LIN {X 0,Y 510.056,Z 394.446,A -85,B 0,C 180,E1 -5580.789,E2 -5580.789} C_VEL
LIN {X 0,Y 509.95,Z 394.463,A -85,B 0,C 180,E1 -5583.16,E2 -5583.16} C_VEL
LIN {X 0,Y 509.969,Z 394.456,A -85,B 0,C 180,E1 -5586.329,E2 -5586.329} C_VEL
LIN {X 0,Y 509.909,Z 394.465,A -85,B 0,C 180,E1 -5588.72,E2 -5588.72} C_VEL
LIN {X 0,Y 509.894,Z 394.466,A -85,B 0,C 180,E1 -5591.931,E2 -5591.931} C_VEL
LIN {X 0,Y 509.883,Z 394.475,A -85,B 0,C 180,E1 -5595.242,E2 -5595.242} C_VEL
LIN {X 0,Y 509.879,Z 394.467,A -85,B 0,C 180,E1 -5598.001,E2 -5598.001} C_VEL
LIN {X 0,Y 509.841,Z 394.479,A -85,B 0,C 180,E1 -5601.002,E2 -5601.002} C_VEL
LIN {X 0,Y 509.86,Z 394.471,A -85,B 0,C 180,E1 -5604.426,E2 -5604.426} C_VEL
LIN {X 0,Y 509.878,Z 394.476,A -85,B 0,C 180,E1 -5607.055,E2 -5607.055} C_VEL
LIN {X 0,Y 509.871,Z 394.469,A -85,B 0,C 180,E1 -5609.75,E2 -5609.75} C_VEL
LIN {X 0,Y 509.868,Z 394.475,A -85,B 0,C 180,E1 -5612.775,E2 -5612.775} C_VEL
LIN {X 0,Y 509.834,Z 394.474,A -85,B 0,C 180,E1 -5615.581,E2 -5615.581} C_VEL
LIN {X 0,Y 509.85,Z 394.473,A -85,B 0,C 180,E1 -5618.337,E2 -5618.337} C_VEL
LIN {X 0,Y 509.857,Z 394.471,A -85,B 0,C 180,E1 -5621.425,E2 -5621.425} C_VEL
LIN {X 0,Y 509.848,Z 394.479,A -85,B 0,C 180,E1 -5624.668,E2 -5624.668} C_VEL
LIN {X 0,Y 509.853,Z 394.472,A -85,B 0,C 180,E1 -5628.103,E2 -5628.103} C_VEL
LIN {X 0,Y 509.84,Z 394.481,A -85,B 0,C 180,E1 -5630.648,E2 -5630.648} C_VEL
LIN {X 0,Y 509.825,Z 394.474,A -85,B 0,C 180,E1 -5633.744,E2 -5633.744} C_VEL
LIN {X 0,Y 509.159,Z 394.564,A -85,B 0,C 180,E1 -5634.404,E2 -5634.404} C_VEL
LIN {X 0,Y 506.341,Z 394.913,A -85,B 0,C 180,E1 -5635.476,E2 -5635.476} C_VEL
LIN {X 0,Y 503.948,Z 395.212,A -85,B 0,C 180,E1 -5636.339,E2 -5636.339} C_VEL
LIN {X 0,Y 502.9,Z 395.34,A -85,B 0,C 180,E1 -5637.006,E2 -5637.006} C_VEL
LIN {X 0,Y 502.803,Z 395.349,A -85,B 0,C 180,E1 -5637.231,E2 -5637.231} C_VEL
LIN {X 0,Y 502.809,Z 395.351,A -85,B 0,C 180,E1 -5640.065,E2 -5640.065} C_VEL
LIN {X 0,Y 502.83,Z 395.353,A -85,B 0,C 180,E1 -5642.534,E2 -5642.534} C_VEL
LIN {X 0,Y 502.824,Z 395.346,A -85,B 0,C 180,E1 -5645.299,E2 -5645.299} C_VEL
LIN {X 0,Y 502.78,Z 395.353,A -85,B 0,C 180,E1 -5647.827,E2 -5647.827} C_VEL
LIN {X 0,Y 502.821,Z 395.355,A -85,B 0,C 180,E1 -5650.4,E2 -5650.4} C_VEL
LIN {X 0,Y 502.83,Z 395.349,A -85,B 0,C 180,E1 -5652.932,E2 -5652.932} C_VEL
LIN {X 0,Y 502.841,Z 395.346,A -85,B 0,C 180,E1 -5655.429,E2 -5655.429} C_VEL
LIN {X 0,Y 502.874,Z 395.344,A -85,B 0,C 180,E1 -5658.717,E2 -5658.717} C_VEL
LIN {X 0,Y 502.898,Z 395.344,A -85,B 0,C 180,E1 -5661.967,E2 -5661.967} C_VEL
LIN {X 0,Y 502.936,Z 395.339,A -85,B 0,C 180,E1 -5664.387,E2 -5664.387} C_VEL
LIN {X 0,Y 503.023,Z 395.327,A -85,B 0,C 180,E1 -5667.598,E2 -5667.598} C_VEL
LIN {X 0,Y 503.025,Z 395.33,A -85,B 0,C 180,E1 -5670,E2 -5670} C_VEL
LIN {X 0,Y 503.023,Z 395.327,A -85,B 0,C 180,E1 -5672.402,E2 -5672.402} C_VEL
LIN {X 0,Y 502.936,Z 395.339,A -85,B 0,C 180,E1 -5675.613,E2 -5675.613} C_VEL
LIN {X 0,Y 502.898,Z 395.344,A -85,B 0,C 180,E1 -5678.033,E2 -5678.033} C_VEL
LIN {X 0,Y 502.874,Z 395.344,A -85,B 0,C 180,E1 -5681.283,E2 -5681.283} C_VEL
LIN {X 0,Y 502.841,Z 395.346,A -85,B 0,C 180,E1 -5684.571,E2 -5684.571} C_VEL
LIN {X 0,Y 502.857,Z 395.35,A -85,B 0,C 180,E1 -5687.907,E2 -5687.907} C_VEL
LIN {X 0,Y 502.824,Z 395.346,A -85,B 0,C 180,E1 -5690.536,E2 -5690.536} C_VEL
LIN {X 0,Y 502.789,Z 395.352,A -85,B 0,C 180,E1 -5693.04,E2 -5693.04} C_VEL
LIN {X 0,Y 502.837,Z 395.352,A -85,B 0,C 180,E1 -5695.675,E2 -5695.675} C_VEL
LIN {X 0,Y 502.835,Z 395.345,A -85,B 0,C 180,E1 -5698.372,E2 -5698.372} C_VEL
LIN {X 0,Y 502.791,Z 395.359,A -85,B 0,C 180,E1 -5701.499,E2 -5701.499} C_VEL
LIN {X 0,Y 502.801,Z 395.349,A -85,B 0,C 180,E1 -5704.444,E2 -5704.444} C_VEL
LIN {X 0,Y 502.774,Z 395.358,A -85,B 0,C 180,E1 -5707.178,E2 -5707.178} C_VEL
LIN {X 0,Y 502.781,Z 395.352,A -85,B 0,C 180,E1 -5710.015,E2 -5710.015} C_VEL
LIN {X 0,Y 502.795,Z 395.35,A -85,B 0,C 180,E1 -5712.199,E2 -5712.199} C_VEL
LIN {X 0,Y 502.792,Z 395.356,A -85,B 0,C 180,E1 -5715.468,E2 -5715.468} C_VEL
LIN {X 0,Y 502.821,Z 395.347,A -85,B 0,C 180,E1 -5717.864,E2 -5717.864} C_VEL
LIN {X 0,Y 502.794,Z 395.356,A -85,B 0,C 180,E1 -5721.024,E2 -5721.024} C_VEL
LIN {X 0,Y 502.777,Z 395.352,A -85,B 0,C 180,E1 -5724.167,E2 -5724.167} C_VEL
LIN {X 0,Y 502.824,Z 395.354,A -85,B 0,C 180,E1 -5726.993,E2 -5726.993} C_VEL
LIN {X 0,Y 502.821,Z 395.346,A -85,B 0,C 180,E1 -5730.062,E2 -5730.062} C_VEL
LIN {X 0,Y 502.826,Z 395.349,A -85,B 0,C 180,E1 -5732.533,E2 -5732.533} C_VEL
LIN {X 0,Y 502.819,Z 395.35,A -85,B 0,C 180,E1 -5735.298,E2 -5735.298} C_VEL
LIN {X 0,Y 502.771,Z 395.353,A -85,B 0,C 180,E1 -5737.827,E2 -5737.827} C_VEL
LIN {X 0,Y 502.816,Z 395.35,A -85,B 0,C 180,E1 -5740.4,E2 -5740.4} C_VEL
LIN {X 0,Y 502.827,Z 395.353,A -85,B 0,C 180,E1 -5742.932,E2 -5742.932} C_VEL
LIN {X 0,Y 502.835,Z 395.346,A -85,B 0,C 180,E1 -5745.429,E2 -5745.429} C_VEL
LIN {X 0,Y 502.868,Z 395.35,A -85,B 0,C 180,E1 -5748.717,E2 -5748.717} C_VEL
LIN {X 0,Y 502.892,Z 395.338,A -85,B 0,C 180,E1 -5751.967,E2 -5751.967} C_VEL
LIN {X 0,Y 502.938,Z 395.337,A -85,B 0,C 180,E1 -5754.387,E2 -5754.387} C_VEL
LIN {X 0,Y 503.016,Z 395.322,A -85,B 0,C 180,E1 -5757.598,E2 -5757.598} C_VEL
LIN {X 0,Y 503.017,Z 395.324,A -85,B 0,C 180,E1 -5760,E2 -5760} C_VEL
LIN {X 0,Y 503.016,Z 395.33,A -85,B 0,C 180,E1 -5762.403,E2 -5762.403} C_VEL
LIN {X 0,Y 502.931,Z 395.333,A -85,B 0,C 180,E1 -5765.614,E2 -5765.614} C_VEL
LIN {X 0,Y 502.894,Z 395.341,A -85,B 0,C 180,E1 -5768.034,E2 -5768.034} C_VEL
LIN {X 0,Y 502.869,Z 395.34,A -85,B 0,C 180,E1 -5771.284,E2 -5771.284} C_VEL
LIN {X 0,Y 502.837,Z 395.349,A -85,B 0,C 180,E1 -5774.571,E2 -5774.571} C_VEL
LIN {X 0,Y 502.854,Z 395.346,A -85,B 0,C 180,E1 -5777.908,E2 -5777.908} C_VEL
LIN {X 0,Y 502.821,Z 395.35,A -85,B 0,C 180,E1 -5780.537,E2 -5780.537} C_VEL
LIN {X 0,Y 502.787,Z 395.351,A -85,B 0,C 180,E1 -5783.041,E2 -5783.041} C_VEL
LIN {X 0,Y 502.834,Z 395.348,A -85,B 0,C 180,E1 -5785.676,E2 -5785.676} C_VEL
LIN {X 0,Y 502.835,Z 395.349,A -85,B 0,C 180,E1 -5788.373,E2 -5788.373} C_VEL
LIN {X 0,Y 502.792,Z 395.352,A -85,B 0,C 180,E1 -5791.501,E2 -5791.501} C_VEL
LIN {X 0,Y 502.801,Z 395.352,A -85,B 0,C 180,E1 -5794.445,E2 -5794.445} C_VEL
LIN {X 0,Y 502.777,Z 395.355,A -85,B 0,C 180,E1 -5797.179,E2 -5797.179} C_VEL
LIN {X 0,Y 502.815,Z 395.356,A -85,B 0,C 180,E1 -5800.013,E2 -5800.013} C_VEL
LIN {X 0,Y 502.772,Z 395.361,A -85,B 0,C 180,E1 -5803.232,E2 -5803.232} C_VEL
LIN {X 0,Y 503.215,Z 398.378,A -85,B 0,C 180,E1 -5805.71,E2 -5805.71} C_VEL
LIN {X 0,Y 503.523,Z 401.387,A -85,B 0,C 180,E1 -5807.937,E2 -5807.937} C_VEL
LIN {X 0,Y 503.395,Z 406.002,A -85,B 0,C 180,E1 -5811.08,E2 -5811.08} C_VEL
LIN {X 0,Y 503.27,Z 409.188,A -85,B 0,C 180,E1 -5813.097,E2 -5813.097} C_VEL
LIN {X 0,Y 503.076,Z 414.026,A -85,B 0,C 180,E1 -5816.028,E2 -5816.028} C_VEL
LIN {X 0,Y 502.905,Z 418.988,A -85,B 0,C 180,E1 -5818.865,E2 -5818.865} C_VEL
LIN {X 0,Y 502.694,Z 424.278,A -85,B 0,C 180,E1 -5821.737,E2 -5821.737} C_VEL
LIN {X 0,Y 502.539,Z 429.165,A -85,B 0,C 180,E1 -5824.309,E2 -5824.309} C_VEL
LIN {X 0,Y 502.429,Z 434.376,A -85,B 0,C 180,E1 -5826.942,E2 -5826.942} C_VEL
LIN {X 0,Y 502.377,Z 439.796,A -85,B 0,C 180,E1 -5829.603,E2 -5829.603} C_VEL
LIN {X 0,Y 502.22,Z 446.73,A -85,B 0,C 180,E1 -5832.911,E2 -5832.911} C_VEL
LIN {X 0,Y 502.208,Z 452.775,A -85,B 0,C 180,E1 -5835.721,E2 -5835.721} C_VEL
LIN {X 0,Y 504.263,Z 465.671,A -85,B 0,C 180,E1 -5836.115,E2 -5836.115} C_VEL
LIN {X 0,Y 504.533,Z 469.583,A -85,B 0,C 180,E1 -5836.251,E2 -5836.251} C_VEL
LIN {X 0,Y 504.232,Z 481.517,A -85,B 0,C 180,E1 -5836.756,E2 -5836.756} C_VEL
LIN {X 0,Y 503.981,Z 490.989,A -85,B 0,C 180,E1 -5837.271,E2 -5837.271} C_VEL
LIN {X 0,Y 503.754,Z 499.544,A -85,B 0,C 180,E1 -5837.836,E2 -5837.836} C_VEL
LIN {X 0,Y 503.436,Z 508.258,A -85,B 0,C 180,E1 -5838.526,E2 -5838.526} C_VEL
LIN {X 0,Y 503.115,Z 516.79,A -85,B 0,C 180,E1 -5839.334,E2 -5839.334} C_VEL
LIN {X 0,Y 502.88,Z 524.011,A -85,B 0,C 180,E1 -5840.143,E2 -5840.143} C_VEL
LIN {X 0,Y 502.663,Z 530.214,A -85,B 0,C 180,E1 -5840.95,E2 -5840.95} C_VEL
LIN {X 0,Y 502.487,Z 536.752,A -85,B 0,C 180,E1 -5841.96,E2 -5841.96} C_VEL
LIN {X 0,Y 502.332,Z 542.306,A -85,B 0,C 180,E1 -5842.989,E2 -5842.989} C_VEL
LIN {X 0,Y 502.237,Z 546.742,A -85,B 0,C 180,E1 -5843.976,E2 -5843.976} C_VEL
LIN {X 0,Y 502.116,Z 551.062,A -85,B 0,C 180,E1 -5845.183,E2 -5845.183} C_VEL
LIN {X 0,Y 502.145,Z 553.427,A -85,B 0,C 180,E1 -5845.987,E2 -5845.987} C_VEL
LIN {X 0,Y 502.121,Z 555.222,A -85,B 0,C 180,E1 -5846.791,E2 -5846.791} C_VEL
LIN {X 0,Y 502.037,Z 557.66,A -85,B 0,C 180,E1 -5848.396,E2 -5848.396} C_VEL
LIN {X 0,Y 501.991,Z 558.246,A -85,B 0,C 180,E1 -5849.198,E2 -5849.198} C_VEL
LIN {X 0,Y 501.991,Z 558.246,A -85,B 0,C 180,E1 -5850.802,E2 -5850.802} C_VEL
LIN {X 0,Y 502.037,Z 557.66,A -85,B 0,C 180,E1 -5851.604,E2 -5851.604} C_VEL
LIN {X 0,Y 502.121,Z 555.222,A -85,B 0,C 180,E1 -5853.209,E2 -5853.209} C_VEL
LIN {X 0,Y 502.115,Z 552.277,A -85,B 0,C 180,E1 -5854.415,E2 -5854.415} C_VEL
LIN {X 0,Y 502.232,Z 548.295,A -85,B 0,C 180,E1 -5855.621,E2 -5855.621} C_VEL
LIN {X 0,Y 502.277,Z 543.359,A -85,B 0,C 180,E1 -5856.79,E2 -5856.79} C_VEL
LIN {X 0,Y 502.418,Z 537.906,A -85,B 0,C 180,E1 -5857.839,E2 -5857.839} C_VEL
LIN {X 0,Y 502.617,Z 531.59,A -85,B 0,C 180,E1 -5858.848,E2 -5858.848} C_VEL
LIN {X 0,Y 502.83,Z 525.639,A -85,B 0,C 180,E1 -5859.655,E2 -5859.655} C_VEL
LIN {X 0,Y 503.039,Z 518.709,A -85,B 0,C 180,E1 -5860.464,E2 -5860.464} C_VEL
LIN {X 0,Y 503.344,Z 510.528,A -85,B 0,C 180,E1 -5861.272,E2 -5861.272} C_VEL
LIN {X 0,Y 503.647,Z 502.014,A -85,B 0,C 180,E1 -5861.98,E2 -5861.98} C_VEL
LIN {X 0,Y 503.838,Z 493.852,A -85,B 0,C 180,E1 -5862.553,E2 -5862.553} C_VEL
LIN {X 0,Y 504.15,Z 484.539,A -85,B 0,C 180,E1 -5863.093,E2 -5863.093} C_VEL
LIN {X 0,Y 504.438,Z 474.736,A -85,B 0,C 180,E1 -5863.546,E2 -5863.546} C_VEL
LIN {X 0,Y 504.476,Z 466.989,A -85,B 0,C 180,E1 -5863.841,E2 -5863.841} C_VEL
LIN {X 0,Y 502.51,Z 454.885,A -85,B 0,C 180,E1 -5864.219,E2 -5864.219} C_VEL
LIN {X 0,Y 502.208,Z 452.775,A -85,B 0,C 180,E1 -5864.279,E2 -5864.279} C_VEL
LIN {X 0,Y 502.22,Z 446.73,A -85,B 0,C 180,E1 -5867.089,E2 -5867.089} C_VEL
LIN {X 0,Y 502.378,Z 439.641,A -85,B 0,C 180,E1 -5870.471,E2 -5870.471} C_VEL
LIN {X 0,Y 502.429,Z 434.376,A -85,B 0,C 180,E1 -5873.058,E2 -5873.058} C_VEL
LIN {X 0,Y 502.538,Z 429.161,A -85,B 0,C 180,E1 -5875.691,E2 -5875.691} C_VEL
LIN {X 0,Y 502.698,Z 424.005,A -85,B 0,C 180,E1 -5878.381,E2 -5878.381} C_VEL
LIN {X 0,Y 502.905,Z 418.961,A -85,B 0,C 180,E1 -5881.135,E2 -5881.135} C_VEL
LIN {X 0,Y 503.077,Z 414.006,A -85,B 0,C 180,E1 -5883.972,E2 -5883.972} C_VEL
LIN {X 0,Y 503.267,Z 409.15,A -85,B 0,C 180,E1 -5886.904,E2 -5886.904} C_VEL
LIN {X 0,Y 503.45,Z 404.431,A -85,B 0,C 180,E1 -5889.951,E2 -5889.951} C_VEL
LIN {X 0,Y 503.494,Z 401.04,A -85,B 0,C 180,E1 -5892.285,E2 -5892.285} C_VEL
LIN {X 0,Y 503.169,Z 398.012,A -85,B 0,C 180,E1 -5894.574,E2 -5894.574} C_VEL
LIN {X 0,Y 502.77,Z 395.359,A -85,B 0,C 180,E1 -5896.768,E2 -5896.768} C_VEL
LIN {X 0,Y 502.815,Z 395.356,A -85,B 0,C 180,E1 -5899.987,E2 -5899.987} C_VEL
LIN {X 0,Y 502.774,Z 395.355,A -85,B 0,C 180,E1 -5903.053,E2 -5903.053} C_VEL
LIN {X 0,Y 502.803,Z 395.358,A -85,B 0,C 180,E1 -5906.006,E2 -5906.006} C_VEL
LIN {X 0,Y 502.794,Z 395.35,A -85,B 0,C 180,E1 -5908.856,E2 -5908.856} C_VEL
LIN {X 0,Y 502.839,Z 395.35,A -85,B 0,C 180,E1 -5911.704,E2 -5911.704} C_VEL
LIN {X 0,Y 502.834,Z 395.348,A -85,B 0,C 180,E1 -5914.324,E2 -5914.324} C_VEL
LIN {X 0,Y 502.798,Z 395.351,A -85,B 0,C 180,E1 -5917.296,E2 -5917.296} C_VEL
LIN {X 0,Y 502.818,Z 395.348,A -85,B 0,C 180,E1 -5920.399,E2 -5920.399} C_VEL
LIN {X 0,Y 502.829,Z 395.346,A -85,B 0,C 180,E1 -5922.931,E2 -5922.931} C_VEL
LIN {X 0,Y 502.837,Z 395.349,A -85,B 0,C 180,E1 -5925.429,E2 -5925.429} C_VEL
LIN {X 0,Y 502.869,Z 395.34,A -85,B 0,C 180,E1 -5928.716,E2 -5928.716} C_VEL
LIN {X 0,Y 502.894,Z 395.341,A -85,B 0,C 180,E1 -5931.966,E2 -5931.966} C_VEL
LIN {X 0,Y 502.931,Z 395.333,A -85,B 0,C 180,E1 -5934.386,E2 -5934.386} C_VEL
LIN {X 0,Y 503.016,Z 395.33,A -85,B 0,C 180,E1 -5937.597,E2 -5937.597} C_VEL
LIN {X 0,Y 503.017,Z 395.324,A -85,B 0,C 180,E1 -5940,E2 -5940} C_VEL
LIN {X 0,Y 503.016,Z 395.322,A -85,B 0,C 180,E1 -5942.402,E2 -5942.402} C_VEL
LIN {X 0,Y 502.938,Z 395.337,A -85,B 0,C 180,E1 -5945.613,E2 -5945.613} C_VEL
LIN {X 0,Y 502.893,Z 395.338,A -85,B 0,C 180,E1 -5948.033,E2 -5948.033} C_VEL
LIN {X 0,Y 502.868,Z 395.35,A -85,B 0,C 180,E1 -5951.283,E2 -5951.283} C_VEL
LIN {X 0,Y 502.835,Z 395.346,A -85,B 0,C 180,E1 -5954.571,E2 -5954.571} C_VEL
LIN {X 0,Y 502.852,Z 395.343,A -85,B 0,C 180,E1 -5957.907,E2 -5957.907} C_VEL
LIN {X 0,Y 502.819,Z 395.348,A -85,B 0,C 180,E1 -5960.536,E2 -5960.536} C_VEL
LIN {X 0,Y 502.784,Z 395.359,A -85,B 0,C 180,E1 -5963.04,E2 -5963.04} C_VEL
LIN {X 0,Y 502.832,Z 395.346,A -85,B 0,C 180,E1 -5965.675,E2 -5965.675} C_VEL
LIN {X 0,Y 502.833,Z 395.346,A -85,B 0,C 180,E1 -5968.373,E2 -5968.373} C_VEL
LIN {X 0,Y 502.788,Z 395.352,A -85,B 0,C 180,E1 -5971.5,E2 -5971.5} C_VEL
LIN {X 0,Y 502.798,Z 395.352,A -85,B 0,C 180,E1 -5974.445,E2 -5974.445} C_VEL
LIN {X 0,Y 502.772,Z 395.357,A -85,B 0,C 180,E1 -5977.179,E2 -5977.179} C_VEL
LIN {X 0,Y 502.818,Z 395.347,A -85,B 0,C 180,E1 -5980.012,E2 -5980.012} C_VEL
LIN {X 0,Y 502.821,Z 395.348,A -85,B 0,C 180,E1 -5982.203,E2 -5982.203} C_VEL
LIN {X 0,Y 502.793,Z 395.35,A -85,B 0,C 180,E1 -5985.468,E2 -5985.468} C_VEL
LIN {X 0,Y 502.822,Z 395.346,A -85,B 0,C 180,E1 -5987.865,E2 -5987.865} C_VEL
LIN {X 0,Y 502.795,Z 395.353,A -85,B 0,C 180,E1 -5991.024,E2 -5991.024} C_VEL
LIN {X 0,Y 502.779,Z 395.355,A -85,B 0,C 180,E1 -5994.168,E2 -5994.168} C_VEL
LIN {X 0,Y 502.803,Z 395.349,A -85,B 0,C 180,E1 -5997.231,E2 -5997.231} C_VEL
LIN {X 0,Y 502.103,Z 395.438,A -85,B 0,C 180,E1 -5997.9,E2 -5997.9} C_VEL
LIN {X 0,Y 499.238,Z 395.795,A -85,B 0,C 180,E1 -5998.986,E2 -5998.986} C_VEL
LIN {X 0,Y 496.842,Z 396.094,A -85,B 0,C 180,E1 -5999.861,E2 -5999.861} C_VEL
LIN {X 0,Y 495.825,Z 396.226,A -85,B 0,C 180,E1 -6000.536,E2 -6000.536} C_VEL
LIN {X 0,Y 495.747,Z 396.228,A -85,B 0,C 180,E1 -6000.765,E2 -6000.765} C_VEL
LIN {X 0,Y 495.794,Z 396.224,A -85,B 0,C 180,E1 -6003.933,E2 -6003.933} C_VEL
LIN {X 0,Y 495.761,Z 396.226,A -85,B 0,C 180,E1 -6007.138,E2 -6007.138} C_VEL
LIN {X 0,Y 495.767,Z 396.231,A -85,B 0,C 180,E1 -6010.11,E2 -6010.11} C_VEL
LIN {X 0,Y 495.782,Z 396.229,A -85,B 0,C 180,E1 -6012.682,E2 -6012.682} C_VEL
LIN {X 0,Y 495.786,Z 396.225,A -85,B 0,C 180,E1 -6015.217,E2 -6015.217} C_VEL
LIN {X 0,Y 495.848,Z 396.221,A -85,B 0,C 180,E1 -6018.555,E2 -6018.555} C_VEL
LIN {X 0,Y 495.869,Z 396.22,A -85,B 0,C 180,E1 -6021.852,E2 -6021.852} C_VEL
LIN {X 0,Y 495.894,Z 396.217,A -85,B 0,C 180,E1 -6024.307,E2 -6024.307} C_VEL
LIN {X 0,Y 495.991,Z 396.202,A -85,B 0,C 180,E1 -6027.564,E2 -6027.564} C_VEL
LIN {X 0,Y 495.996,Z 396.206,A -85,B 0,C 180,E1 -6030,E2 -6030} C_VEL
LIN {X 0,Y 495.991,Z 396.202,A -85,B 0,C 180,E1 -6032.436,E2 -6032.436} C_VEL
LIN {X 0,Y 495.893,Z 396.217,A -85,B 0,C 180,E1 -6035.693,E2 -6035.693} C_VEL
LIN {X 0,Y 495.869,Z 396.22,A -85,B 0,C 180,E1 -6038.148,E2 -6038.148} C_VEL
LIN {X 0,Y 495.848,Z 396.221,A -85,B 0,C 180,E1 -6041.445,E2 -6041.445} C_VEL
LIN {X 0,Y 495.786,Z 396.225,A -85,B 0,C 180,E1 -6044.783,E2 -6044.783} C_VEL
LIN {X 0,Y 495.782,Z 396.229,A -85,B 0,C 180,E1 -6047.318,E2 -6047.318} C_VEL
LIN {X 0,Y 495.767,Z 396.231,A -85,B 0,C 180,E1 -6049.89,E2 -6049.89} C_VEL
LIN {X 0,Y 495.756,Z 396.227,A -85,B 0,C 180,E1 -6052.861,E2 -6052.861} C_VEL
LIN {X 0,Y 495.794,Z 396.224,A -85,B 0,C 180,E1 -6056.067,E2 -6056.067} C_VEL
LIN {X 0,Y 495.766,Z 396.226,A -85,B 0,C 180,E1 -6058.814,E2 -6058.814} C_VEL
LIN {X 0,Y 495.753,Z 396.232,A -85,B 0,C 180,E1 -6061.726,E2 -6061.726} C_VEL
LIN {X 0,Y 495.77,Z 396.225,A -85,B 0,C 180,E1 -6064.695,E2 -6064.695} C_VEL
LIN {X 0,Y 495.725,Z 396.237,A -85,B 0,C 180,E1 -6067.561,E2 -6067.561} C_VEL
LIN {X 0,Y 495.759,Z 396.227,A -85,B 0,C 180,E1 -6070.699,E2 -6070.699} C_VEL
LIN {X 0,Y 495.727,Z 396.233,A -85,B 0,C 180,E1 -6073.695,E2 -6073.695} C_VEL
LIN {X 0,Y 495.726,Z 396.23,A -85,B 0,C 180,E1 -6076.304,E2 -6076.304} C_VEL
LIN {X 0,Y 495.758,Z 396.234,A -85,B 0,C 180,E1 -6079.3,E2 -6079.3} C_VEL
LIN {X 0,Y 495.722,Z 396.231,A -85,B 0,C 180,E1 -6082.438,E2 -6082.438} C_VEL
LIN {X 0,Y 495.777,Z 396.228,A -85,B 0,C 180,E1 -6085.457,E2 -6085.457} C_VEL
LIN {X 0,Y 495.75,Z 396.228,A -85,B 0,C 180,E1 -6088.364,E2 -6088.364} C_VEL
LIN {X 0,Y 495.781,Z 396.226,A -85,B 0,C 180,E1 -6091.506,E2 -6091.506} C_VEL
LIN {X 0,Y 495.79,Z 396.222,A -85,B 0,C 180,E1 -6093.933,E2 -6093.933} C_VEL
LIN {X 0,Y 495.751,Z 396.232,A -85,B 0,C 180,E1 -6097.139,E2 -6097.139} C_VEL
LIN {X 0,Y 495.768,Z 396.226,A -85,B 0,C 180,E1 -6100.11,E2 -6100.11} C_VEL
LIN {X 0,Y 495.779,Z 396.23,A -85,B 0,C 180,E1 -6102.682,E2 -6102.682} C_VEL
LIN {X 0,Y 495.78,Z 396.226,A -85,B 0,C 180,E1 -6105.217,E2 -6105.217} C_VEL
LIN {X 0,Y 495.842,Z 396.222,A -85,B 0,C 180,E1 -6108.555,E2 -6108.555} C_VEL
LIN {X 0,Y 495.863,Z 396.213,A -85,B 0,C 180,E1 -6111.852,E2 -6111.852} C_VEL
LIN {X 0,Y 495.894,Z 396.213,A -85,B 0,C 180,E1 -6114.307,E2 -6114.307} C_VEL
LIN {X 0,Y 495.985,Z 396.198,A -85,B 0,C 180,E1 -6117.564,E2 -6117.564} C_VEL
LIN {X 0,Y 495.989,Z 396.199,A -85,B 0,C 180,E1 -6120,E2 -6120} C_VEL
LIN {X 0,Y 495.985,Z 396.206,A -85,B 0,C 180,E1 -6122.437,E2 -6122.437} C_VEL
LIN {X 0,Y 495.888,Z 396.211,A -85,B 0,C 180,E1 -6125.694,E2 -6125.694} C_VEL
LIN {X 0,Y 495.865,Z 396.218,A -85,B 0,C 180,E1 -6128.149,E2 -6128.149} C_VEL
LIN {X 0,Y 495.843,Z 396.216,A -85,B 0,C 180,E1 -6131.446,E2 -6131.446} C_VEL
LIN {X 0,Y 495.782,Z 396.226,A -85,B 0,C 180,E1 -6134.784,E2 -6134.784} C_VEL
LIN {X 0,Y 495.78,Z 396.223,A -85,B 0,C 180,E1 -6137.319,E2 -6137.319} C_VEL
LIN {X 0,Y 495.764,Z 396.23,A -85,B 0,C 180,E1 -6139.891,E2 -6139.891} C_VEL
LIN {X 0,Y 495.754,Z 396.228,A -85,B 0,C 180,E1 -6142.862,E2 -6142.862} C_VEL
LIN {X 0,Y 495.785,Z 396.231,A -85,B 0,C 180,E1 -6146.069,E2 -6146.069} C_VEL
LIN {X 0,Y 495.773,Z 396.225,A -85,B 0,C 180,E1 -6148.815,E2 -6148.815} C_VEL
LIN {X 0,Y 495.754,Z 396.231,A -85,B 0,C 180,E1 -6151.727,E2 -6151.727} C_VEL
LIN {X 0,Y 495.771,Z 396.225,A -85,B 0,C 180,E1 -6154.696,E2 -6154.696} C_VEL
LIN {X 0,Y 495.728,Z 396.237,A -85,B 0,C 180,E1 -6157.562,E2 -6157.562} C_VEL
LIN {X 0,Y 495.773,Z 396.23,A -85,B 0,C 180,E1 -6160.7,E2 -6160.7} C_VEL
LIN {X 0,Y 495.724,Z 396.238,A -85,B 0,C 180,E1 -6162.884,E2 -6162.884} C_VEL
LIN {X 0,Y 496.099,Z 398.79,A -85,B 0,C 180,E1 -6165.099,E2 -6165.099} C_VEL
LIN {X 0,Y 496.467,Z 401.787,A -85,B 0,C 180,E1 -6167.402,E2 -6167.402} C_VEL
LIN {X 0,Y 496.431,Z 405.287,A -85,B 0,C 180,E1 -6169.861,E2 -6169.861} C_VEL
LIN {X 0,Y 496.309,Z 409.246,A -85,B 0,C 180,E1 -6172.491,E2 -6172.491} C_VEL
LIN {X 0,Y 496.064,Z 414.086,A -85,B 0,C 180,E1 -6175.48,E2 -6175.48} C_VEL
LIN {X 0,Y 495.903,Z 418.991,A -85,B 0,C 180,E1 -6178.375,E2 -6178.375} C_VEL
LIN {X 0,Y 495.661,Z 424.68,A -85,B 0,C 180,E1 -6181.535,E2 -6181.535} C_VEL
LIN {X 0,Y 495.497,Z 429.124,A -85,B 0,C 180,E1 -6183.916,E2 -6183.916} C_VEL
LIN {X 0,Y 495.354,Z 434.3,A -85,B 0,C 180,E1 -6186.594,E2 -6186.594} C_VEL
LIN {X 0,Y 495.294,Z 440.055,A -85,B 0,C 180,E1 -6189.474,E2 -6189.474} C_VEL
LIN {X 0,Y 495.159,Z 446.593,A -85,B 0,C 180,E1 -6192.659,E2 -6192.659} C_VEL
LIN {X 0,Y 495.097,Z 452.675,A -85,B 0,C 180,E1 -6195.525,E2 -6195.525} C_VEL
LIN {X 0,Y 496.754,Z 462.831,A -85,B 0,C 180,E1 -6195.822,E2 -6195.822} C_VEL
LIN {X 0,Y 497.657,Z 469.386,A -85,B 0,C 180,E1 -6196.057,E2 -6196.057} C_VEL
LIN {X 0,Y 497.307,Z 481.319,A -85,B 0,C 180,E1 -6196.568,E2 -6196.568} C_VEL
LIN {X 0,Y 497.033,Z 491.084,A -85,B 0,C 180,E1 -6197.108,E2 -6197.108} C_VEL
LIN {X 0,Y 496.767,Z 499.197,A -85,B 0,C 180,E1 -6197.651,E2 -6197.651} C_VEL
LIN {X 0,Y 496.453,Z 508.06,A -85,B 0,C 180,E1 -6198.362,E2 -6198.362} C_VEL
LIN {X 0,Y 496.117,Z 516.592,A -85,B 0,C 180,E1 -6199.182,E2 -6199.182} C_VEL
LIN {X 0,Y 495.853,Z 523.813,A -85,B 0,C 180,E1 -6200.002,E2 -6200.002} C_VEL
LIN {X 0,Y 495.628,Z 530.016,A -85,B 0,C 180,E1 -6200.821,E2 -6200.821} C_VEL
LIN {X 0,Y 495.416,Z 536.554,A -85,B 0,C 180,E1 -6201.845,E2 -6201.845} C_VEL
LIN {X 0,Y 495.273,Z 541.055,A -85,B 0,C 180,E1 -6202.663,E2 -6202.663} C_VEL
LIN {X 0,Y 495.137,Z 547.054,A -85,B 0,C 180,E1 -6204.023,E2 -6204.023} C_VEL
LIN {X 0,Y 495.043,Z 550.865,A -85,B 0,C 180,E1 -6205.114,E2 -6205.114} C_VEL
LIN {X 0,Y 495.04,Z 553.229,A -85,B 0,C 180,E1 -6205.93,E2 -6205.93} C_VEL
LIN {X 0,Y 495.043,Z 555.026,A -85,B 0,C 180,E1 -6206.745,E2 -6206.745} C_VEL
LIN {X 0,Y 494.963,Z 557.464,A -85,B 0,C 180,E1 -6208.373,E2 -6208.373} C_VEL
LIN {X 0,Y 494.911,Z 558.05,A -85,B 0,C 180,E1 -6209.186,E2 -6209.186} C_VEL
LIN {X 0,Y 494.911,Z 558.05,A -85,B 0,C 180,E1 -6210.814,E2 -6210.814} C_VEL
LIN {X 0,Y 494.963,Z 557.464,A -85,B 0,C 180,E1 -6211.627,E2 -6211.627} C_VEL
LIN {X 0,Y 495.043,Z 555.026,A -85,B 0,C 180,E1 -6213.255,E2 -6213.255} C_VEL
LIN {X 0,Y 495.019,Z 552.08,A -85,B 0,C 180,E1 -6214.478,E2 -6214.478} C_VEL
LIN {X 0,Y 495.148,Z 548.098,A -85,B 0,C 180,E1 -6215.702,E2 -6215.702} C_VEL
LIN {X 0,Y 495.219,Z 542.97,A -85,B 0,C 180,E1 -6216.928,E2 -6216.928} C_VEL
LIN {X 0,Y 495.368,Z 537.709,A -85,B 0,C 180,E1 -6217.951,E2 -6217.951} C_VEL
LIN {X 0,Y 495.578,Z 531.392,A -85,B 0,C 180,E1 -6218.974,E2 -6218.974} C_VEL
LIN {X 0,Y 495.782,Z 525.44,A -85,B 0,C 180,E1 -6219.794,E2 -6219.794} C_VEL
LIN {X 0,Y 496.023,Z 518.511,A -85,B 0,C 180,E1 -6220.614,E2 -6220.614} C_VEL
LIN {X 0,Y 496.365,Z 510.33,A -85,B 0,C 180,E1 -6221.433,E2 -6221.433} C_VEL
LIN {X 0,Y 496.669,Z 501.816,A -85,B 0,C 180,E1 -6222.151,E2 -6222.151} C_VEL
LIN {X 0,Y 496.87,Z 494.194,A -85,B 0,C 180,E1 -6222.698,E2 -6222.698} C_VEL
LIN {X 0,Y 497.195,Z 484.341,A -85,B 0,C 180,E1 -6223.279,E2 -6223.279} C_VEL
LIN {X 0,Y 497.531,Z 474.539,A -85,B 0,C 180,E1 -6223.738,E2 -6223.738} C_VEL
LIN {X 0,Y 497.455,Z 467.224,A -85,B 0,C 180,E1 -6224.027,E2 -6224.027} C_VEL
LIN {X 0,Y 495.441,Z 454.862,A -85,B 0,C 180,E1 -6224.422,E2 -6224.422} C_VEL
LIN {X 0,Y 495.085,Z 452.613,A -85,B 0,C 180,E1 -6224.489,E2 -6224.489} C_VEL
LIN {X 0,Y 495.159,Z 446.593,A -85,B 0,C 180,E1 -6227.341,E2 -6227.341} C_VEL
LIN {X 0,Y 495.305,Z 439.546,A -85,B 0,C 180,E1 -6230.776,E2 -6230.776} C_VEL
LIN {X 0,Y 495.354,Z 434.298,A -85,B 0,C 180,E1 -6233.406,E2 -6233.406} C_VEL
LIN {X 0,Y 495.497,Z 429.118,A -85,B 0,C 180,E1 -6236.084,E2 -6236.084} C_VEL
LIN {X 0,Y 495.678,Z 423.992,A -85,B 0,C 180,E1 -6238.82,E2 -6238.82} C_VEL
LIN {X 0,Y 495.899,Z 418.767,A -85,B 0,C 180,E1 -6241.751,E2 -6241.751} C_VEL
LIN {X 0,Y 496.082,Z 413.661,A -85,B 0,C 180,E1 -6244.745,E2 -6244.745} C_VEL
LIN {X 0,Y 496.315,Z 409.197,A -85,B 0,C 180,E1 -6247.535,E2 -6247.535} C_VEL
LIN {X 0,Y 496.456,Z 404.525,A -85,B 0,C 180,E1 -6250.63,E2 -6250.63} C_VEL
LIN {X 0,Y 496.447,Z 401.49,A -85,B 0,C 180,E1 -6252.805,E2 -6252.805} C_VEL
LIN {X 0,Y 496.059,Z 398.533,A -85,B 0,C 180,E1 -6255.102,E2 -6255.102} C_VEL
LIN {X 0,Y 495.723,Z 396.238,A -85,B 0,C 180,E1 -6257.116,E2 -6257.116} C_VEL
LIN {X 0,Y 495.783,Z 396.231,A -85,B 0,C 180,E1 -6259.948,E2 -6259.948} C_VEL
LIN {X 0,Y 495.727,Z 396.236,A -85,B 0,C 180,E1 -6262.552,E2 -6262.552} C_VEL
LIN {X 0,Y 495.78,Z 396.228,A -85,B 0,C 180,E1 -6265.456,E2 -6265.456} C_VEL
LIN {X 0,Y 495.754,Z 396.23,A -85,B 0,C 180,E1 -6268.363,E2 -6268.363} C_VEL
LIN {X 0,Y 495.784,Z 396.226,A -85,B 0,C 180,E1 -6271.505,E2 -6271.505} C_VEL
LIN {X 0,Y 495.785,Z 396.231,A -85,B 0,C 180,E1 -6273.931,E2 -6273.931} C_VEL
LIN {X 0,Y 495.754,Z 396.228,A -85,B 0,C 180,E1 -6277.138,E2 -6277.138} C_VEL
LIN {X 0,Y 495.764,Z 396.23,A -85,B 0,C 180,E1 -6280.109,E2 -6280.109} C_VEL
LIN {X 0,Y 495.78,Z 396.223,A -85,B 0,C 180,E1 -6282.681,E2 -6282.681} C_VEL
LIN {X 0,Y 495.782,Z 396.226,A -85,B 0,C 180,E1 -6285.216,E2 -6285.216} C_VEL
LIN {X 0,Y 495.843,Z 396.216,A -85,B 0,C 180,E1 -6288.554,E2 -6288.554} C_VEL
LIN {X 0,Y 495.865,Z 396.218,A -85,B 0,C 180,E1 -6291.851,E2 -6291.851} C_VEL
LIN {X 0,Y 495.888,Z 396.211,A -85,B 0,C 180,E1 -6294.306,E2 -6294.306} C_VEL
LIN {X 0,Y 495.985,Z 396.206,A -85,B 0,C 180,E1 -6297.563,E2 -6297.563} C_VEL
LIN {X 0,Y 495.989,Z 396.199,A -85,B 0,C 180,E1 -6300,E2 -6300} C_VEL
LIN {X 0,Y 495.985,Z 396.198,A -85,B 0,C 180,E1 -6302.436,E2 -6302.436} C_VEL
LIN {X 0,Y 495.895,Z 396.213,A -85,B 0,C 180,E1 -6305.693,E2 -6305.693} C_VEL
LIN {X 0,Y 495.864,Z 396.213,A -85,B 0,C 180,E1 -6308.148,E2 -6308.148} C_VEL
LIN {X 0,Y 495.842,Z 396.222,A -85,B 0,C 180,E1 -6311.445,E2 -6311.445} C_VEL
LIN {X 0,Y 495.78,Z 396.226,A -85,B 0,C 180,E1 -6314.783,E2 -6314.783} C_VEL
LIN {X 0,Y 495.779,Z 396.23,A -85,B 0,C 180,E1 -6317.318,E2 -6317.318} C_VEL
LIN {X 0,Y 495.768,Z 396.226,A -85,B 0,C 180,E1 -6319.89,E2 -6319.89} C_VEL
LIN {X 0,Y 495.751,Z 396.232,A -85,B 0,C 180,E1 -6322.861,E2 -6322.861} C_VEL
LIN {X 0,Y 495.79,Z 396.222,A -85,B 0,C 180,E1 -6326.067,E2 -6326.067} C_VEL
LIN {X 0,Y 495.771,Z 396.231,A -85,B 0,C 180,E1 -6328.814,E2 -6328.814} C_VEL
LIN {X 0,Y 495.75,Z 396.228,A -85,B 0,C 180,E1 -6331.726,E2 -6331.726} C_VEL
LIN {X 0,Y 495.768,Z 396.231,A -85,B 0,C 180,E1 -6334.696,E2 -6334.696} C_VEL
LIN {X 0,Y 495.724,Z 396.231,A -85,B 0,C 180,E1 -6337.561,E2 -6337.561} C_VEL
LIN {X 0,Y 495.785,Z 396.223,A -85,B 0,C 180,E1 -6340.052,E2 -6340.052} C_VEL
LIN {X 0,Y 495.755,Z 396.234,A -85,B 0,C 180,E1 -6342.879,E2 -6342.879} C_VEL
LIN {X 0,Y 495.729,Z 396.231,A -85,B 0,C 180,E1 -6346,E2 -6346} C_VEL
LIN {X 0,Y 495.756,Z 396.235,A -85,B 0,C 180,E1 -6348.706,E2 -6348.706} C_VEL
LIN {X 0,Y 495.744,Z 396.229,A -85,B 0,C 180,E1 -6351.409,E2 -6351.409} C_VEL
LIN {X 0,Y 495.751,Z 396.234,A -85,B 0,C 180,E1 -6354.463,E2 -6354.463} C_VEL
LIN {X 0,Y 495.764,Z 396.226,A -85,B 0,C 180,E1 -6357.406,E2 -6357.406} C_VEL
LIN {X 0,Y 495.761,Z 396.231,A -85,B 0,C 180,E1 -6360.254,E2 -6360.254} C_VEL
LIN {X 0,Y 495.747,Z 396.228,A -85,B 0,C 180,E1 -6360.765,E2 -6360.765} C_VEL
LIN {X 0,Y 495.092,Z 396.311,A -85,B 0,C 180,E1 -6361.444,E2 -6361.444} C_VEL
LIN {X 0,Y 492.239,Z 396.672,A -85,B 0,C 180,E1 -6362.547,E2 -6362.547} C_VEL
LIN {X 0,Y 489.832,Z 396.968,A -85,B 0,C 180,E1 -6363.436,E2 -6363.436} C_VEL
LIN {X 0,Y 488.815,Z 397.096,A -85,B 0,C 180,E1 -6364.122,E2 -6364.122} C_VEL
LIN {X 0,Y 488.742,Z 397.107,A -85,B 0,C 180,E1 -6364.354,E2 -6364.354} C_VEL
LIN {X 0,Y 488.723,Z 397.103,A -85,B 0,C 180,E1 -6367.154,E2 -6367.154} C_VEL
LIN {X 0,Y 488.721,Z 397.105,A -85,B 0,C 180,E1 -6369.811,E2 -6369.811} C_VEL
LIN {X 0,Y 488.73,Z 397.109,A -85,B 0,C 180,E1 -6372.424,E2 -6372.424} C_VEL
LIN {X 0,Y 488.758,Z 397.101,A -85,B 0,C 180,E1 -6375,E2 -6375} C_VEL
LIN {X 0,Y 488.802,Z 397.1,A -85,B 0,C 180,E1 -6378.388,E2 -6378.388} C_VEL
LIN {X 0,Y 488.814,Z 397.098,A -85,B 0,C 180,E1 -6381.734,E2 -6381.734} C_VEL
LIN {X 0,Y 488.853,Z 397.094,A -85,B 0,C 180,E1 -6384.224,E2 -6384.224} C_VEL
LIN {X 0,Y 488.959,Z 397.078,A -85,B 0,C 180,E1 -6387.529,E2 -6387.529} C_VEL
LIN {X 0,Y 488.951,Z 397.078,A -85,B 0,C 180,E1 -6390.824,E2 -6390.824} C_VEL
LIN {X 0,Y 488.959,Z 397.078,A -85,B 0,C 180,E1 -6392.471,E2 -6392.471} C_VEL
LIN {X 0,Y 488.853,Z 397.094,A -85,B 0,C 180,E1 -6395.776,E2 -6395.776} C_VEL
LIN {X 0,Y 488.814,Z 397.098,A -85,B 0,C 180,E1 -6398.266,E2 -6398.266} C_VEL
LIN {X 0,Y 488.802,Z 397.1,A -85,B 0,C 180,E1 -6401.612,E2 -6401.612} C_VEL
LIN {X 0,Y 488.758,Z 397.101,A -85,B 0,C 180,E1 -6405,E2 -6405} C_VEL
LIN {X 0,Y 488.75,Z 397.102,A -85,B 0,C 180,E1 -6408.442,E2 -6408.442} C_VEL
LIN {X 0,Y 488.702,Z 397.107,A -85,B 0,C 180,E1 -6411.07,E2 -6411.07} C_VEL
LIN {X 0,Y 488.688,Z 397.114,A -85,B 0,C 180,E1 -6413.745,E2 -6413.745} C_VEL
LIN {X 0,Y 488.794,Z 397.095,A -85,B 0,C 180,E1 -6416.945,E2 -6416.945} C_VEL
LIN {X 0,Y 488.704,Z 397.105,A -85,B 0,C 180,E1 -6420.363,E2 -6420.363} C_VEL
LIN {X 0,Y 488.73,Z 397.11,A -85,B 0,C 180,E1 -6423.484,E2 -6423.484} C_VEL
LIN {X 0,Y 488.682,Z 397.108,A -85,B 0,C 180,E1 -6426.355,E2 -6426.355} C_VEL
LIN {X 0,Y 488.694,Z 397.113,A -85,B 0,C 180,E1 -6429.254,E2 -6429.254} C_VEL
LIN {X 0,Y 488.716,Z 397.108,A -85,B 0,C 180,E1 -6431.602,E2 -6431.602} C_VEL
LIN {X 0,Y 488.704,Z 397.108,A -85,B 0,C 180,E1 -6434.801,E2 -6434.801} C_VEL
LIN {X 0,Y 488.687,Z 397.112,A -85,B 0,C 180,E1 -6437.475,E2 -6437.475} C_VEL
LIN {X 0,Y 488.724,Z 397.105,A -85,B 0,C 180,E1 -6439.676,E2 -6439.676} C_VEL
LIN {X 0,Y 488.674,Z 397.113,A -85,B 0,C 180,E1 -6442.841,E2 -6442.841} C_VEL
LIN {X 0,Y 488.726,Z 397.103,A -85,B 0,C 180,E1 -6445.887,E2 -6445.887} C_VEL
LIN {X 0,Y 488.687,Z 397.113,A -85,B 0,C 180,E1 -6448.821,E2 -6448.821} C_VEL
LIN {X 0,Y 488.737,Z 397.102,A -85,B 0,C 180,E1 -6451.671,E2 -6451.671} C_VEL
LIN {X 0,Y 488.741,Z 397.103,A -85,B 0,C 180,E1 -6454.445,E2 -6454.445} C_VEL
LIN {X 0,Y 488.714,Z 397.109,A -85,B 0,C 180,E1 -6457.153,E2 -6457.153} C_VEL
LIN {X 0,Y 488.719,Z 397.103,A -85,B 0,C 180,E1 -6459.811,E2 -6459.811} C_VEL
LIN {X 0,Y 488.725,Z 397.106,A -85,B 0,C 180,E1 -6462.424,E2 -6462.424} C_VEL
LIN {X 0,Y 488.752,Z 397.104,A -85,B 0,C 180,E1 -6465,E2 -6465} C_VEL
LIN {X 0,Y 488.796,Z 397.098,A -85,B 0,C 180,E1 -6468.388,E2 -6468.388} C_VEL
LIN {X 0,Y 488.808,Z 397.092,A -85,B 0,C 180,E1 -6471.734,E2 -6471.734} C_VEL
LIN {X 0,Y 488.852,Z 397.09,A -85,B 0,C 180,E1 -6474.225,E2 -6474.225} C_VEL
LIN {X 0,Y 488.953,Z 397.074,A -85,B 0,C 180,E1 -6477.529,E2 -6477.529} C_VEL
LIN {X 0,Y 488.946,Z 397.079,A -85,B 0,C 180,E1 -6480.824,E2 -6480.824} C_VEL
LIN {X 0,Y 488.953,Z 397.083,A -85,B 0,C 180,E1 -6482.472,E2 -6482.472} C_VEL
LIN {X 0,Y 488.847,Z 397.088,A -85,B 0,C 180,E1 -6485.776,E2 -6485.776} C_VEL
LIN {X 0,Y 488.81,Z 397.099,A -85,B 0,C 180,E1 -6488.267,E2 -6488.267} C_VEL
LIN {X 0,Y 488.797,Z 397.094,A -85,B 0,C 180,E1 -6491.613,E2 -6491.613} C_VEL
LIN {X 0,Y 488.754,Z 397.099,A -85,B 0,C 180,E1 -6495.001,E2 -6495.001} C_VEL
LIN {X 0,Y 488.747,Z 397.105,A -85,B 0,C 180,E1 -6498.443,E2 -6498.443} C_VEL
LIN {X 0,Y 488.699,Z 397.106,A -85,B 0,C 180,E1 -6501.072,E2 -6501.072} C_VEL
LIN {X 0,Y 488.686,Z 397.11,A -85,B 0,C 180,E1 -6503.746,E2 -6503.746} C_VEL
LIN {X 0,Y 488.786,Z 397.095,A -85,B 0,C 180,E1 -6506.945,E2 -6506.945} C_VEL
LIN {X 0,Y 488.713,Z 397.108,A -85,B 0,C 180,E1 -6510.366,E2 -6510.366} C_VEL
LIN {X 0,Y 488.731,Z 397.104,A -85,B 0,C 180,E1 -6513.485,E2 -6513.485} C_VEL
LIN {X 0,Y 488.685,Z 397.113,A -85,B 0,C 180,E1 -6516.357,E2 -6516.357} C_VEL
LIN {X 0,Y 488.737,Z 397.106,A -85,B 0,C 180,E1 -6519.251,E2 -6519.251} C_VEL
LIN {X 0,Y 488.706,Z 397.113,A -85,B 0,C 180,E1 -6521.601,E2 -6521.601} C_VEL
LIN {X 0,Y 488.707,Z 397.254,A -85,B 0,C 180,E1 -6522.827,E2 -6522.827} C_VEL
LIN {X 0,Y 489.255,Z 400.997,A -85,B 0,C 180,E1 -6525.909,E2 -6525.909} C_VEL
LIN {X 0,Y 489.494,Z 404.157,A -85,B 0,C 180,E1 -6528.297,E2 -6528.297} C_VEL
LIN {X 0,Y 489.364,Z 407.815,A -85,B 0,C 180,E1 -6530.853,E2 -6530.853} C_VEL
LIN {X 0,Y 489.179,Z 411.961,A -85,B 0,C 180,E1 -6533.567,E2 -6533.567} C_VEL
LIN {X 0,Y 488.964,Z 416.668,A -85,B 0,C 180,E1 -6536.476,E2 -6536.476} C_VEL
LIN {X 0,Y 488.76,Z 422.324,A -85,B 0,C 180,E1 -6539.784,E2 -6539.784} C_VEL
LIN {X 0,Y 488.516,Z 428.354,A -85,B 0,C 180,E1 -6543.121,E2 -6543.121} C_VEL
LIN {X 0,Y 488.305,Z 434.23,A -85,B 0,C 180,E1 -6546.235,E2 -6546.235} C_VEL
LIN {X 0,Y 488.216,Z 440.296,A -85,B 0,C 180,E1 -6549.341,E2 -6549.341} C_VEL
LIN {X 0,Y 488.069,Z 446.456,A -85,B 0,C 180,E1 -6552.399,E2 -6552.399} C_VEL
LIN {X 0,Y 488.028,Z 452.452,A -85,B 0,C 180,E1 -6555.297,E2 -6555.297} C_VEL
LIN {X 0,Y 490.37,Z 467.021,A -85,B 0,C 180,E1 -6555.766,E2 -6555.766} C_VEL
LIN {X 0,Y 490.667,Z 471.765,A -85,B 0,C 180,E1 -6555.96,E2 -6555.96} C_VEL
LIN {X 0,Y 490.357,Z 482.129,A -85,B 0,C 180,E1 -6556.427,E2 -6556.427} C_VEL
LIN {X 0,Y 490.069,Z 491.155,A -85,B 0,C 180,E1 -6556.939,E2 -6556.939} C_VEL
LIN {X 0,Y 489.755,Z 500.266,A -85,B 0,C 180,E1 -6557.57,E2 -6557.57} C_VEL
LIN {X 0,Y 489.431,Z 508.997,A -85,B 0,C 180,E1 -6558.298,E2 -6558.298} C_VEL
LIN {X 0,Y 489.129,Z 516.394,A -85,B 0,C 180,E1 -6559.025,E2 -6559.025} C_VEL
LIN {X 0,Y 488.829,Z 523.615,A -85,B 0,C 180,E1 -6559.856,E2 -6559.856} C_VEL
LIN {X 0,Y 488.58,Z 529.818,A -85,B 0,C 180,E1 -6560.687,E2 -6560.687} C_VEL
LIN {X 0,Y 488.35,Z 536.356,A -85,B 0,C 180,E1 -6561.726,E2 -6561.726} C_VEL
LIN {X 0,Y 488.203,Z 540.857,A -85,B 0,C 180,E1 -6562.556,E2 -6562.556} C_VEL
LIN {X 0,Y 488.038,Z 546.263,A -85,B 0,C 180,E1 -6563.778,E2 -6563.778} C_VEL
LIN {X 0,Y 487.973,Z 550.668,A -85,B 0,C 180,E1 -6565.043,E2 -6565.043} C_VEL
LIN {X 0,Y 487.936,Z 553.031,A -85,B 0,C 180,E1 -6565.87,E2 -6565.87} C_VEL
LIN {X 0,Y 487.966,Z 554.829,A -85,B 0,C 180,E1 -6566.697,E2 -6566.697} C_VEL
LIN {X 0,Y 487.891,Z 557.268,A -85,B 0,C 180,E1 -6568.349,E2 -6568.349} C_VEL
LIN {X 0,Y 487.834,Z 557.853,A -85,B 0,C 180,E1 -6569.175,E2 -6569.175} C_VEL
LIN {X 0,Y 487.834,Z 557.853,A -85,B 0,C 180,E1 -6570.825,E2 -6570.825} C_VEL
LIN {X 0,Y 487.891,Z 557.268,A -85,B 0,C 180,E1 -6571.651,E2 -6571.651} C_VEL
LIN {X 0,Y 487.966,Z 554.829,A -85,B 0,C 180,E1 -6573.303,E2 -6573.303} C_VEL
LIN {X 0,Y 487.931,Z 551.883,A -85,B 0,C 180,E1 -6574.544,E2 -6574.544} C_VEL
LIN {X 0,Y 488.045,Z 547.9,A -85,B 0,C 180,E1 -6575.785,E2 -6575.785} C_VEL
LIN {X 0,Y 488.1,Z 544.687,A -85,B 0,C 180,E1 -6576.614,E2 -6576.614} C_VEL
LIN {X 0,Y 488.262,Z 538.666,A -85,B 0,C 180,E1 -6577.859,E2 -6577.859} C_VEL
LIN {X 0,Y 488.474,Z 532.57,A -85,B 0,C 180,E1 -6578.897,E2 -6578.897} C_VEL
LIN {X 0,Y 488.705,Z 526.87,A -85,B 0,C 180,E1 -6579.728,E2 -6579.728} C_VEL
LIN {X 0,Y 489.024,Z 518.313,A -85,B 0,C 180,E1 -6580.768,E2 -6580.768} C_VEL
LIN {X 0,Y 489.392,Z 510.133,A -85,B 0,C 180,E1 -6581.598,E2 -6581.598} C_VEL
LIN {X 0,Y 489.686,Z 501.618,A -85,B 0,C 180,E1 -6582.326,E2 -6582.326} C_VEL
LIN {X 0,Y 489.958,Z 493.387,A -85,B 0,C 180,E1 -6582.92,E2 -6582.92} C_VEL
LIN {X 0,Y 490.276,Z 484.143,A -85,B 0,C 180,E1 -6583.47,E2 -6583.47} C_VEL
LIN {X 0,Y 490.628,Z 474.342,A -85,B 0,C 180,E1 -6583.935,E2 -6583.935} C_VEL
LIN {X 0,Y 490.499,Z 467.821,A -85,B 0,C 180,E1 -6584.203,E2 -6584.203} C_VEL
LIN {X 0,Y 488.393,Z 454.983,A -85,B 0,C 180,E1 -6584.629,E2 -6584.629} C_VEL
LIN {X 0,Y 488.028,Z 452.452,A -85,B 0,C 180,E1 -6584.703,E2 -6584.703} C_VEL
LIN {X 0,Y 488.096,Z 445.376,A -85,B 0,C 180,E1 -6588.135,E2 -6588.135} C_VEL
LIN {X 0,Y 488.234,Z 439.438,A -85,B 0,C 180,E1 -6591.092,E2 -6591.092} C_VEL
LIN {X 0,Y 488.305,Z 434.221,A -85,B 0,C 180,E1 -6593.765,E2 -6593.765} C_VEL
LIN {X 0,Y 488.506,Z 428.351,A -85,B 0,C 180,E1 -6596.877,E2 -6596.877} C_VEL
LIN {X 0,Y 488.759,Z 422.321,A -85,B 0,C 180,E1 -6600.216,E2 -6600.216} C_VEL
LIN {X 0,Y 488.964,Z 416.654,A -85,B 0,C 180,E1 -6603.524,E2 -6603.524} C_VEL
LIN {X 0,Y 489.187,Z 411.949,A -85,B 0,C 180,E1 -6606.434,E2 -6606.434} C_VEL
LIN {X 0,Y 489.364,Z 407.737,A -85,B 0,C 180,E1 -6609.19,E2 -6609.19} C_VEL
LIN {X 0,Y 489.502,Z 404.132,A -85,B 0,C 180,E1 -6611.704,E2 -6611.704} C_VEL
LIN {X 0,Y 489.254,Z 400.974,A -85,B 0,C 180,E1 -6614.09,E2 -6614.09} C_VEL
LIN {X 0,Y 488.706,Z 397.256,A -85,B 0,C 180,E1 -6617.173,E2 -6617.173} C_VEL
LIN {X 0,Y 488.729,Z 397.108,A -85,B 0,C 180,E1 -6619.676,E2 -6619.676} C_VEL
LIN {X 0,Y 488.676,Z 397.117,A -85,B 0,C 180,E1 -6622.277,E2 -6622.277} C_VEL
LIN {X 0,Y 488.724,Z 397.106,A -85,B 0,C 180,E1 -6625.051,E2 -6625.051} C_VEL
LIN {X 0,Y 488.702,Z 397.113,A -85,B 0,C 180,E1 -6628.044,E2 -6628.044} C_VEL
LIN {X 0,Y 488.728,Z 397.102,A -85,B 0,C 180,E1 -6630.73,E2 -6630.73} C_VEL
LIN {X 0,Y 488.751,Z 397.103,A -85,B 0,C 180,E1 -6633.527,E2 -6633.527} C_VEL
LIN {X 0,Y 488.686,Z 397.11,A -85,B 0,C 180,E1 -6636.254,E2 -6636.254} C_VEL
LIN {X 0,Y 488.739,Z 397.102,A -85,B 0,C 180,E1 -6639.175,E2 -6639.175} C_VEL
LIN {X 0,Y 488.727,Z 397.103,A -85,B 0,C 180,E1 -6642.423,E2 -6642.423} C_VEL
LIN {X 0,Y 488.754,Z 397.099,A -85,B 0,C 180,E1 -6644.999,E2 -6644.999} C_VEL
LIN {X 0,Y 488.797,Z 397.094,A -85,B 0,C 180,E1 -6648.387,E2 -6648.387} C_VEL
LIN {X 0,Y 488.81,Z 397.099,A -85,B 0,C 180,E1 -6651.733,E2 -6651.733} C_VEL
LIN {X 0,Y 488.847,Z 397.088,A -85,B 0,C 180,E1 -6654.224,E2 -6654.224} C_VEL
LIN {X 0,Y 488.953,Z 397.083,A -85,B 0,C 180,E1 -6657.528,E2 -6657.528} C_VEL
LIN {X 0,Y 488.946,Z 397.076,A -85,B 0,C 180,E1 -6660.823,E2 -6660.823} C_VEL
LIN {X 0,Y 488.953,Z 397.074,A -85,B 0,C 180,E1 -6662.471,E2 -6662.471} C_VEL
LIN {X 0,Y 488.852,Z 397.09,A -85,B 0,C 180,E1 -6665.775,E2 -6665.775} C_VEL
LIN {X 0,Y 488.809,Z 397.092,A -85,B 0,C 180,E1 -6668.266,E2 -6668.266} C_VEL
LIN {X 0,Y 488.796,Z 397.098,A -85,B 0,C 180,E1 -6671.612,E2 -6671.612} C_VEL
LIN {X 0,Y 488.752,Z 397.104,A -85,B 0,C 180,E1 -6675,E2 -6675} C_VEL
LIN {X 0,Y 488.745,Z 397.101,A -85,B 0,C 180,E1 -6678.442,E2 -6678.442} C_VEL
LIN {X 0,Y 488.697,Z 397.114,A -85,B 0,C 180,E1 -6681.071,E2 -6681.071} C_VEL
LIN {X 0,Y 488.683,Z 397.109,A -85,B 0,C 180,E1 -6683.745,E2 -6683.745} C_VEL
LIN {X 0,Y 488.789,Z 397.102,A -85,B 0,C 180,E1 -6686.945,E2 -6686.945} C_VEL
LIN {X 0,Y 488.71,Z 397.106,A -85,B 0,C 180,E1 -6690.365,E2 -6690.365} C_VEL
LIN {X 0,Y 488.727,Z 397.104,A -85,B 0,C 180,E1 -6693.485,E2 -6693.485} C_VEL
LIN {X 0,Y 488.68,Z 397.11,A -85,B 0,C 180,E1 -6696.356,E2 -6696.356} C_VEL
LIN {X 0,Y 488.74,Z 397.103,A -85,B 0,C 180,E1 -6699.25,E2 -6699.25} C_VEL
LIN {X 0,Y 488.727,Z 397.107,A -85,B 0,C 180,E1 -6702.521,E2 -6702.521} C_VEL
LIN {X 0,Y 488.694,Z 397.107,A -85,B 0,C 180,E1 -6705.976,E2 -6705.976} C_VEL
LIN {X 0,Y 488.712,Z 397.111,A -85,B 0,C 180,E1 -6708.586,E2 -6708.586} C_VEL
LIN {X 0,Y 488.674,Z 397.109,A -85,B 0,C 180,E1 -6711.8,E2 -6711.8} C_VEL
LIN {X 0,Y 488.722,Z 397.105,A -85,B 0,C 180,E1 -6715.052,E2 -6715.052} C_VEL
LIN {X 0,Y 488.7,Z 397.108,A -85,B 0,C 180,E1 -6718.046,E2 -6718.046} C_VEL
LIN {X 0,Y 488.717,Z 397.108,A -85,B 0,C 180,E1 -6720.763,E2 -6720.763} C_VEL
LIN {X 0,Y 488.761,Z 397.098,A -85,B 0,C 180,E1 -6723.529,E2 -6723.529} C_VEL
LIN {X 0,Y 488.742,Z 397.107,A -85,B 0,C 180,E1 -6724.354,E2 -6724.354} C_VEL
LIN {X 0,Y 488.095,Z 397.194,A -85,B 0,C 180,E1 -6725.042,E2 -6725.042} C_VEL
LIN {X 0,Y 485.226,Z 397.549,A -85,B 0,C 180,E1 -6726.158,E2 -6726.158} C_VEL
LIN {X 0,Y 482.78,Z 397.847,A -85,B 0,C 180,E1 -6727.058,E2 -6727.058} C_VEL
LIN {X 0,Y 481.722,Z 397.976,A -85,B 0,C 180,E1 -6727.754,E2 -6727.754} C_VEL
LIN {X 0,Y 481.633,Z 397.987,A -85,B 0,C 180,E1 -6727.989,E2 -6727.989} C_VEL
LIN {X 0,Y 481.701,Z 397.986,A -85,B 0,C 180,E1 -6730.393,E2 -6730.393} C_VEL
LIN {X 0,Y 481.687,Z 397.982,A -85,B 0,C 180,E1 -6733.034,E2 -6733.034} C_VEL
LIN {X 0,Y 481.686,Z 397.983,A -85,B 0,C 180,E1 -6735.639,E2 -6735.639} C_VEL
LIN {X 0,Y 481.747,Z 397.979,A -85,B 0,C 180,E1 -6738.215,E2 -6738.215} C_VEL
LIN {X 0,Y 481.759,Z 397.976,A -85,B 0,C 180,E1 -6741.612,E2 -6741.612} C_VEL
LIN {X 0,Y 481.814,Z 397.971,A -85,B 0,C 180,E1 -6744.14,E2 -6744.14} C_VEL
LIN {X 0,Y 481.926,Z 397.954,A -85,B 0,C 180,E1 -6747.493,E2 -6747.493} C_VEL
LIN {X 0,Y 481.902,Z 397.956,A -85,B 0,C 180,E1 -6750.836,E2 -6750.836} C_VEL
LIN {X 0,Y 481.926,Z 397.954,A -85,B 0,C 180,E1 -6752.507,E2 -6752.507} C_VEL
LIN {X 0,Y 481.814,Z 397.971,A -85,B 0,C 180,E1 -6755.86,E2 -6755.86} C_VEL
LIN {X 0,Y 481.759,Z 397.976,A -85,B 0,C 180,E1 -6758.388,E2 -6758.388} C_VEL
LIN {X 0,Y 481.747,Z 397.979,A -85,B 0,C 180,E1 -6761.785,E2 -6761.785} C_VEL
LIN {X 0,Y 481.738,Z 397.977,A -85,B 0,C 180,E1 -6765.224,E2 -6765.224} C_VEL
LIN {X 0,Y 481.707,Z 397.979,A -85,B 0,C 180,E1 -6768.721,E2 -6768.721} C_VEL
LIN {X 0,Y 481.641,Z 397.99,A -85,B 0,C 180,E1 -6771.394,E2 -6771.394} C_VEL
LIN {X 0,Y 481.672,Z 397.983,A -85,B 0,C 180,E1 -6774.113,E2 -6774.113} C_VEL
LIN {X 0,Y 481.747,Z 397.975,A -85,B 0,C 180,E1 -6777.14,E2 -6777.14} C_VEL
LIN {X 0,Y 481.673,Z 397.986,A -85,B 0,C 180,E1 -6779.741,E2 -6779.741} C_VEL
LIN {X 0,Y 481.667,Z 397.982,A -85,B 0,C 180,E1 -6782.674,E2 -6782.674} C_VEL
LIN {X 0,Y 481.636,Z 397.99,A -85,B 0,C 180,E1 -6785.709,E2 -6785.709} C_VEL
LIN {X 0,Y 481.664,Z 397.984,A -85,B 0,C 180,E1 -6788.859,E2 -6788.859} C_VEL
LIN {X 0,Y 481.655,Z 397.985,A -85,B 0,C 180,E1 -6791.914,E2 -6791.914} C_VEL
LIN {X 0,Y 481.652,Z 397.984,A -85,B 0,C 180,E1 -6794.457,E2 -6794.457} C_VEL
LIN {X 0,Y 481.669,Z 397.985,A -85,B 0,C 180,E1 -6796.847,E2 -6796.847} C_VEL
LIN {X 0,Y 481.668,Z 397.982,A -85,B 0,C 180,E1 -6800.059,E2 -6800.059} C_VEL
LIN {X 0,Y 481.621,Z 397.994,A -85,B 0,C 180,E1 -6803.253,E2 -6803.253} C_VEL
LIN {X 0,Y 481.7,Z 397.978,A -85,B 0,C 180,E1 -6806.33,E2 -6806.33} C_VEL
LIN {X 0,Y 481.649,Z 397.987,A -85,B 0,C 180,E1 -6809.416,E2 -6809.416} C_VEL
LIN {X 0,Y 481.693,Z 397.979,A -85,B 0,C 180,E1 -6812.168,E2 -6812.168} C_VEL
LIN {X 0,Y 481.709,Z 397.985,A -85,B 0,C 180,E1 -6814.97,E2 -6814.97} C_VEL
LIN {X 0,Y 481.64,Z 397.985,A -85,B 0,C 180,E1 -6817.705,E2 -6817.705} C_VEL
LIN {X 0,Y 481.698,Z 397.98,A -85,B 0,C 180,E1 -6820.393,E2 -6820.393} C_VEL
LIN {X 0,Y 481.682,Z 397.985,A -85,B 0,C 180,E1 -6823.034,E2 -6823.034} C_VEL
LIN {X 0,Y 481.681,Z 397.98,A -85,B 0,C 180,E1 -6825.639,E2 -6825.639} C_VEL
LIN {X 0,Y 481.741,Z 397.975,A -85,B 0,C 180,E1 -6828.215,E2 -6828.215} C_VEL
LIN {X 0,Y 481.753,Z 397.971,A -85,B 0,C 180,E1 -6831.612,E2 -6831.612} C_VEL
LIN {X 0,Y 481.812,Z 397.966,A -85,B 0,C 180,E1 -6834.14,E2 -6834.14} C_VEL
LIN {X 0,Y 481.92,Z 397.95,A -85,B 0,C 180,E1 -6837.493,E2 -6837.493} C_VEL
LIN {X 0,Y 481.897,Z 397.957,A -85,B 0,C 180,E1 -6840.836,E2 -6840.836} C_VEL
LIN {X 0,Y 481.92,Z 397.959,A -85,B 0,C 180,E1 -6842.508,E2 -6842.508} C_VEL
LIN {X 0,Y 481.808,Z 397.966,A -85,B 0,C 180,E1 -6845.861,E2 -6845.861} C_VEL
LIN {X 0,Y 481.755,Z 397.979,A -85,B 0,C 180,E1 -6848.389,E2 -6848.389} C_VEL
LIN {X 0,Y 481.742,Z 397.974,A -85,B 0,C 180,E1 -6851.786,E2 -6851.786} C_VEL
LIN {X 0,Y 481.735,Z 397.973,A -85,B 0,C 180,E1 -6855.225,E2 -6855.225} C_VEL
LIN {X 0,Y 481.705,Z 397.979,A -85,B 0,C 180,E1 -6858.722,E2 -6858.722} C_VEL
LIN {X 0,Y 481.638,Z 397.986,A -85,B 0,C 180,E1 -6861.396,E2 -6861.396} C_VEL
LIN {X 0,Y 481.67,Z 397.99,A -85,B 0,C 180,E1 -6864.114,E2 -6864.114} C_VEL
LIN {X 0,Y 481.741,Z 397.972,A -85,B 0,C 180,E1 -6867.14,E2 -6867.14} C_VEL
LIN {X 0,Y 481.682,Z 397.984,A -85,B 0,C 180,E1 -6869.741,E2 -6869.741} C_VEL
LIN {X 0,Y 481.668,Z 397.982,A -85,B 0,C 180,E1 -6872.675,E2 -6872.675} C_VEL
LIN {X 0,Y 481.638,Z 397.99,A -85,B 0,C 180,E1 -6875.71,E2 -6875.71} C_VEL
LIN {X 0,Y 481.709,Z 397.983,A -85,B 0,C 180,E1 -6879.355,E2 -6879.355} C_VEL
LIN {X 0,Y 481.645,Z 397.992,A -85,B 0,C 180,E1 -6882.161,E2 -6882.161} C_VEL
LIN {X 0,Y 482.013,Z 400.333,A -85,B 0,C 180,E1 -6884.417,E2 -6884.417} C_VEL
LIN {X 0,Y 482.403,Z 403.256,A -85,B 0,C 180,E1 -6886.787,E2 -6886.787} C_VEL
LIN {X 0,Y 482.442,Z 406.575,A -85,B 0,C 180,E1 -6889.246,E2 -6889.246} C_VEL
LIN {X 0,Y 482.259,Z 410.968,A -85,B 0,C 180,E1 -6892.262,E2 -6892.262} C_VEL
LIN {X 0,Y 482.005,Z 415.756,A -85,B 0,C 180,E1 -6895.345,E2 -6895.345} C_VEL
LIN {X 0,Y 481.782,Z 420.664,A -85,B 0,C 180,E1 -6898.322,E2 -6898.322} C_VEL
LIN {X 0,Y 481.576,Z 425.66,A -85,B 0,C 180,E1 -6901.211,E2 -6901.211} C_VEL
LIN {X 0,Y 481.376,Z 430.735,A -85,B 0,C 180,E1 -6904.025,E2 -6904.025} C_VEL
LIN {X 0,Y 481.204,Z 436.195,A -85,B 0,C 180,E1 -6906.944,E2 -6906.944} C_VEL
LIN {X 0,Y 481.128,Z 441.081,A -85,B 0,C 180,E1 -6909.478,E2 -6909.478} C_VEL
LIN {X 0,Y 480.997,Z 446.319,A -85,B 0,C 180,E1 -6912.132,E2 -6912.132} C_VEL
LIN {X 0,Y 480.978,Z 452.291,A -85,B 0,C 180,E1 -6915.077,E2 -6915.077} C_VEL
LIN {X 0,Y 483.344,Z 467.23,A -85,B 0,C 180,E1 -6915.568,E2 -6915.568} C_VEL
LIN {X 0,Y 483.763,Z 471.567,A -85,B 0,C 180,E1 -6915.756,E2 -6915.756} C_VEL
LIN {X 0,Y 483.463,Z 481.932,A -85,B 0,C 180,E1 -6916.229,E2 -6916.229} C_VEL
LIN {X 0,Y 483.136,Z 491.072,A -85,B 0,C 180,E1 -6916.756,E2 -6916.756} C_VEL
LIN {X 0,Y 482.785,Z 500.068,A -85,B 0,C 180,E1 -6917.388,E2 -6917.388} C_VEL
LIN {X 0,Y 482.458,Z 508.8,A -85,B 0,C 180,E1 -6918.126,E2 -6918.126} C_VEL
LIN {X 0,Y 482.147,Z 516.197,A -85,B 0,C 180,E1 -6918.864,E2 -6918.864} C_VEL
LIN {X 0,Y 481.791,Z 523.417,A -85,B 0,C 180,E1 -6919.707,E2 -6919.707} C_VEL
LIN {X 0,Y 481.526,Z 529.619,A -85,B 0,C 180,E1 -6920.55,E2 -6920.55} C_VEL
LIN {X 0,Y 481.309,Z 536.158,A -85,B 0,C 180,E1 -6921.604,E2 -6921.604} C_VEL
LIN {X 0,Y 481.137,Z 540.659,A -85,B 0,C 180,E1 -6922.446,E2 -6922.446} C_VEL
LIN {X 0,Y 480.939,Z 546.522,A -85,B 0,C 180,E1 -6923.809,E2 -6923.809} C_VEL
LIN {X 0,Y 480.905,Z 550.471,A -85,B 0,C 180,E1 -6924.97,E2 -6924.97} C_VEL
LIN {X 0,Y 480.836,Z 552.834,A -85,B 0,C 180,E1 -6925.809,E2 -6925.809} C_VEL
LIN {X 0,Y 480.89,Z 554.632,A -85,B 0,C 180,E1 -6926.649,E2 -6926.649} C_VEL
LIN {X 0,Y 480.793,Z 557.071,A -85,B 0,C 180,E1 -6928.325,E2 -6928.325} C_VEL
LIN {X 0,Y 480.76,Z 557.657,A -85,B 0,C 180,E1 -6929.162,E2 -6929.162} C_VEL
LIN {X 0,Y 480.76,Z 557.657,A -85,B 0,C 180,E1 -6930.838,E2 -6930.838} C_VEL
LIN {X 0,Y 480.793,Z 557.071,A -85,B 0,C 180,E1 -6931.675,E2 -6931.675} C_VEL
LIN {X 0,Y 480.89,Z 554.632,A -85,B 0,C 180,E1 -6933.351,E2 -6933.351} C_VEL
LIN {X 0,Y 480.848,Z 551.685,A -85,B 0,C 180,E1 -6934.611,E2 -6934.611} C_VEL
LIN {X 0,Y 480.947,Z 547.702,A -85,B 0,C 180,E1 -6935.871,E2 -6935.871} C_VEL
LIN {X 0,Y 481.016,Z 544.489,A -85,B 0,C 180,E1 -6936.712,E2 -6936.712} C_VEL
LIN {X 0,Y 481.21,Z 538.469,A -85,B 0,C 180,E1 -6937.975,E2 -6937.975} C_VEL
LIN {X 0,Y 481.423,Z 532.372,A -85,B 0,C 180,E1 -6939.029,E2 -6939.029} C_VEL
LIN {X 0,Y 481.678,Z 526.672,A -85,B 0,C 180,E1 -6939.871,E2 -6939.871} C_VEL
LIN {X 0,Y 482.037,Z 518.116,A -85,B 0,C 180,E1 -6940.926,E2 -6940.926} C_VEL
LIN {X 0,Y 482.421,Z 509.935,A -85,B 0,C 180,E1 -6941.768,E2 -6941.768} C_VEL
LIN {X 0,Y 482.687,Z 502.797,A -85,B 0,C 180,E1 -6942.399,E2 -6942.399} C_VEL
LIN {X 0,Y 483.016,Z 493.19,A -85,B 0,C 180,E1 -6943.109,E2 -6943.109} C_VEL
LIN {X 0,Y 483.414,Z 482.939,A -85,B 0,C 180,E1 -6943.718,E2 -6943.718} C_VEL
LIN {X 0,Y 483.756,Z 472.856,A -85,B 0,C 180,E1 -6944.191,E2 -6944.191} C_VEL
LIN {X 0,Y 483.426,Z 467.618,A -85,B 0,C 180,E1 -6944.416,E2 -6944.416} C_VEL
LIN {X 0,Y 481.362,Z 454.799,A -85,B 0,C 180,E1 -6944.847,E2 -6944.847} C_VEL
LIN {X 0,Y 480.978,Z 452.291,A -85,B 0,C 180,E1 -6944.923,E2 -6944.923} C_VEL
LIN {X 0,Y 481.012,Z 445.563,A -85,B 0,C 180,E1 -6948.248,E2 -6948.248} C_VEL
LIN {X 0,Y 481.144,Z 439.327,A -85,B 0,C 180,E1 -6951.418,E2 -6951.418} C_VEL
LIN {X 0,Y 481.262,Z 434.149,A -85,B 0,C 180,E1 -6954.135,E2 -6954.135} C_VEL
LIN {X 0,Y 481.467,Z 428.727,A -85,B 0,C 180,E1 -6957.073,E2 -6957.073} C_VEL
LIN {X 0,Y 481.632,Z 423.973,A -85,B 0,C 180,E1 -6959.744,E2 -6959.744} C_VEL
LIN {X 0,Y 481.853,Z 418.988,A -85,B 0,C 180,E1 -6962.66,E2 -6962.66} C_VEL
LIN {X 0,Y 482.094,Z 414.142,A -85,B 0,C 180,E1 -6965.67,E2 -6965.67} C_VEL
LIN {X 0,Y 482.304,Z 409.364,A -85,B 0,C 180,E1 -6968.797,E2 -6968.797} C_VEL
LIN {X 0,Y 482.454,Z 406.272,A -85,B 0,C 180,E1 -6970.958,E2 -6970.958} C_VEL
LIN {X 0,Y 482.395,Z 403.204,A -85,B 0,C 180,E1 -6973.243,E2 -6973.243} C_VEL
LIN {X 0,Y 481.984,Z 400.281,A -85,B 0,C 180,E1 -6975.6,E2 -6975.6} C_VEL
LIN {X 0,Y 481.645,Z 397.991,A -85,B 0,C 180,E1 -6977.838,E2 -6977.838} C_VEL
LIN {X 0,Y 481.709,Z 397.983,A -85,B 0,C 180,E1 -6980.645,E2 -6980.645} C_VEL
LIN {X 0,Y 481.638,Z 397.994,A -85,B 0,C 180,E1 -6984.29,E2 -6984.29} C_VEL
LIN {X 0,Y 481.668,Z 397.982,A -85,B 0,C 180,E1 -6987.325,E2 -6987.325} C_VEL
LIN {X 0,Y 481.683,Z 397.984,A -85,B 0,C 180,E1 -6990.259,E2 -6990.259} C_VEL
LIN {X 0,Y 481.739,Z 397.973,A -85,B 0,C 180,E1 -6993.111,E2 -6993.111} C_VEL
LIN {X 0,Y 481.67,Z 397.99,A -85,B 0,C 180,E1 -6995.886,E2 -6995.886} C_VEL
LIN {X 0,Y 481.695,Z 397.979,A -85,B 0,C 180,E1 -6999.027,E2 -6999.027} C_VEL
LIN {X 0,Y 481.7,Z 397.981,A -85,B 0,C 180,E1 -7002.158,E2 -7002.158} C_VEL
LIN {X 0,Y 481.735,Z 397.973,A -85,B 0,C 180,E1 -7004.775,E2 -7004.775} C_VEL
LIN {X 0,Y 481.742,Z 397.974,A -85,B 0,C 180,E1 -7008.214,E2 -7008.214} C_VEL
LIN {X 0,Y 481.755,Z 397.979,A -85,B 0,C 180,E1 -7011.611,E2 -7011.611} C_VEL
LIN {X 0,Y 481.808,Z 397.966,A -85,B 0,C 180,E1 -7014.139,E2 -7014.139} C_VEL
LIN {X 0,Y 481.92,Z 397.959,A -85,B 0,C 180,E1 -7017.492,E2 -7017.492} C_VEL
LIN {X 0,Y 481.897,Z 397.954,A -85,B 0,C 180,E1 -7020.835,E2 -7020.835} C_VEL
LIN {X 0,Y 481.92,Z 397.95,A -85,B 0,C 180,E1 -7022.507,E2 -7022.507} C_VEL
LIN {X 0,Y 481.812,Z 397.966,A -85,B 0,C 180,E1 -7025.86,E2 -7025.86} C_VEL
LIN {X 0,Y 481.754,Z 397.971,A -85,B 0,C 180,E1 -7028.388,E2 -7028.388} C_VEL
LIN {X 0,Y 481.741,Z 397.975,A -85,B 0,C 180,E1 -7031.785,E2 -7031.785} C_VEL
LIN {X 0,Y 481.732,Z 397.982,A -85,B 0,C 180,E1 -7035.224,E2 -7035.224} C_VEL
LIN {X 0,Y 481.703,Z 397.98,A -85,B 0,C 180,E1 -7038.722,E2 -7038.722} C_VEL
LIN {X 0,Y 481.636,Z 397.99,A -85,B 0,C 180,E1 -7041.395,E2 -7041.395} C_VEL
LIN {X 0,Y 481.667,Z 397.982,A -85,B 0,C 180,E1 -7044.113,E2 -7044.113} C_VEL
LIN {X 0,Y 481.743,Z 397.979,A -85,B 0,C 180,E1 -7047.141,E2 -7047.141} C_VEL
LIN {X 0,Y 481.679,Z 397.981,A -85,B 0,C 180,E1 -7049.74,E2 -7049.74} C_VEL
LIN {X 0,Y 481.664,Z 397.987,A -85,B 0,C 180,E1 -7052.674,E2 -7052.674} C_VEL
LIN {X 0,Y 481.634,Z 397.986,A -85,B 0,C 180,E1 -7055.709,E2 -7055.709} C_VEL
LIN {X 0,Y 481.711,Z 397.978,A -85,B 0,C 180,E1 -7059.355,E2 -7059.355} C_VEL
LIN {X 0,Y 481.666,Z 397.983,A -85,B 0,C 180,E1 -7062.158,E2 -7062.158} C_VEL
LIN {X 0,Y 481.652,Z 397.988,A -85,B 0,C 180,E1 -7064.457,E2 -7064.457} C_VEL
LIN {X 0,Y 481.646,Z 397.984,A -85,B 0,C 180,E1 -7067.84,E2 -7067.84} C_VEL
LIN {X 0,Y 481.673,Z 397.99,A -85,B 0,C 180,E1 -7070.651,E2 -7070.651} C_VEL
LIN {X 0,Y 481.625,Z 397.987,A -85,B 0,C 180,E1 -7073.376,E2 -7073.376} C_VEL
LIN {X 0,Y 481.703,Z 397.983,A -85,B 0,C 180,E1 -7076.33,E2 -7076.33} C_VEL
LIN {X 0,Y 481.645,Z 397.984,A -85,B 0,C 180,E1 -7079.417,E2 -7079.417} C_VEL
LIN {X 0,Y 481.696,Z 397.982,A -85,B 0,C 180,E1 -7082.169,E2 -7082.169} C_VEL
LIN {X 0,Y 481.713,Z 397.978,A -85,B 0,C 180,E1 -7084.97,E2 -7084.97} C_VEL
LIN {X 0,Y 481.633,Z 397.987,A -85,B 0,C 180,E1 -7087.989,E2 -7087.989} C_VEL
LIN {X 0,Y 480.965,Z 398.075,A -85,B 0,C 180,E1 -7088.687,E2 -7088.687} C_VEL
LIN {X 0,Y 478.137,Z 398.424,A -85,B 0,C 180,E1 -7089.821,E2 -7089.821} C_VEL
LIN {X 0,Y 475.752,Z 398.724,A -85,B 0,C 180,E1 -7090.736,E2 -7090.736} C_VEL
LIN {X 0,Y 474.732,Z 398.849,A -85,B 0,C 180,E1 -7091.442,E2 -7091.442} C_VEL
LIN {X 0,Y 474.651,Z 398.86,A -85,B 0,C 180,E1 -7091.68,E2 -7091.68} C_VEL
LIN {X 0,Y 474.696,Z 398.857,A -85,B 0,C 180,E1 -7094.545,E2 -7094.545} C_VEL
LIN {X 0,Y 474.701,Z 398.858,A -85,B 0,C 180,E1 -7098.038,E2 -7098.038} C_VEL
LIN {X 0,Y 474.724,Z 398.851,A -85,B 0,C 180,E1 -7101.487,E2 -7101.487} C_VEL
LIN {X 0,Y 474.776,Z 398.848,A -85,B 0,C 180,E1 -7104.053,E2 -7104.053} C_VEL
LIN {X 0,Y 474.892,Z 398.83,A -85,B 0,C 180,E1 -7107.455,E2 -7107.455} C_VEL
LIN {X 0,Y 474.909,Z 398.832,A -85,B 0,C 180,E1 -7110,E2 -7110} C_VEL
LIN {X 0,Y 474.892,Z 398.83,A -85,B 0,C 180,E1 -7112.545,E2 -7112.545} C_VEL
LIN {X 0,Y 474.776,Z 398.848,A -85,B 0,C 180,E1 -7115.947,E2 -7115.947} C_VEL
LIN {X 0,Y 474.724,Z 398.851,A -85,B 0,C 180,E1 -7118.513,E2 -7118.513} C_VEL
LIN {X 0,Y 474.701,Z 398.858,A -85,B 0,C 180,E1 -7121.962,E2 -7121.962} C_VEL
LIN {X 0,Y 474.696,Z 398.857,A -85,B 0,C 180,E1 -7125.455,E2 -7125.455} C_VEL
LIN {X 0,Y 474.66,Z 398.858,A -85,B 0,C 180,E1 -7129.01,E2 -7129.01} C_VEL
LIN {X 0,Y 474.585,Z 398.871,A -85,B 0,C 180,E1 -7131.729,E2 -7131.729} C_VEL
LIN {X 0,Y 474.654,Z 398.855,A -85,B 0,C 180,E1 -7134.493,E2 -7134.493} C_VEL
LIN {X 0,Y 474.693,Z 398.856,A -85,B 0,C 180,E1 -7137.338,E2 -7137.338} C_VEL
LIN {X 0,Y 474.599,Z 398.863,A -85,B 0,C 180,E1 -7140.81,E2 -7140.81} C_VEL
LIN {X 0,Y 474.632,Z 398.86,A -85,B 0,C 180,E1 -7143.984,E2 -7143.984} C_VEL
LIN {X 0,Y 474.568,Z 398.868,A -85,B 0,C 180,E1 -7146.9,E2 -7146.9} C_VEL
LIN {X 0,Y 474.62,Z 398.864,A -85,B 0,C 180,E1 -7149.647,E2 -7149.647} C_VEL
LIN {X 0,Y 474.628,Z 398.862,A -85,B 0,C 180,E1 -7152.932,E2 -7152.932} C_VEL
LIN {X 0,Y 474.607,Z 398.862,A -85,B 0,C 180,E1 -7155.896,E2 -7155.896} C_VEL
LIN {X 0,Y 474.623,Z 398.865,A -85,B 0,C 180,E1 -7159.04,E2 -7159.04} C_VEL
LIN {X 0,Y 474.602,Z 398.864,A -85,B 0,C 180,E1 -7161.704,E2 -7161.704} C_VEL
LIN {X 0,Y 474.621,Z 398.863,A -85,B 0,C 180,E1 -7164.726,E2 -7164.726} C_VEL
LIN {X 0,Y 474.628,Z 398.859,A -85,B 0,C 180,E1 -7167.788,E2 -7167.788} C_VEL
LIN {X 0,Y 474.623,Z 398.866,A -85,B 0,C 180,E1 -7170.883,E2 -7170.883} C_VEL
LIN {X 0,Y 474.657,Z 398.856,A -85,B 0,C 180,E1 -7173.629,E2 -7173.629} C_VEL
LIN {X 0,Y 474.626,Z 398.863,A -85,B 0,C 180,E1 -7176.641,E2 -7176.641} C_VEL
LIN {X 0,Y 474.647,Z 398.857,A -85,B 0,C 180,E1 -7180.09,E2 -7180.09} C_VEL
LIN {X 0,Y 474.642,Z 398.865,A -85,B 0,C 180,E1 -7182.775,E2 -7182.775} C_VEL
LIN {X 0,Y 474.639,Z 398.858,A -85,B 0,C 180,E1 -7185.421,E2 -7185.421} C_VEL
LIN {X 0,Y 474.694,Z 398.851,A -85,B 0,C 180,E1 -7188.038,E2 -7188.038} C_VEL
LIN {X 0,Y 474.719,Z 398.848,A -85,B 0,C 180,E1 -7191.487,E2 -7191.487} C_VEL
LIN {X 0,Y 474.774,Z 398.842,A -85,B 0,C 180,E1 -7194.053,E2 -7194.053} C_VEL
LIN {X 0,Y 474.886,Z 398.827,A -85,B 0,C 180,E1 -7197.456,E2 -7197.456} C_VEL
LIN {X 0,Y 474.902,Z 398.826,A -85,B 0,C 180,E1 -7200,E2 -7200} C_VEL
LIN {X 0,Y 474.886,Z 398.834,A -85,B 0,C 180,E1 -7202.545,E2 -7202.545} C_VEL
LIN {X 0,Y 474.771,Z 398.843,A -85,B 0,C 180,E1 -7205.948,E2 -7205.948} C_VEL
LIN {X 0,Y 474.72,Z 398.854,A -85,B 0,C 180,E1 -7208.514,E2 -7208.514} C_VEL
LIN {X 0,Y 474.696,Z 398.853,A -85,B 0,C 180,E1 -7211.963,E2 -7211.963} C_VEL
LIN {X 0,Y 474.694,Z 398.852,A -85,B 0,C 180,E1 -7215.778,E2 -7215.778} C_VEL
LIN {X 0,Y 474.657,Z 398.855,A -85,B 0,C 180,E1 -7219.011,E2 -7219.011} C_VEL
LIN {X 0,Y 474.582,Z 398.867,A -85,B 0,C 180,E1 -7221.73,E2 -7221.73} C_VEL
LIN {X 0,Y 474.652,Z 398.859,A -85,B 0,C 180,E1 -7224.494,E2 -7224.494} C_VEL
LIN {X 0,Y 474.675,Z 398.853,A -85,B 0,C 180,E1 -7227.335,E2 -7227.335} C_VEL
LIN {X 0,Y 474.608,Z 398.867,A -85,B 0,C 180,E1 -7230.23,E2 -7230.23} C_VEL
LIN {X 0,Y 474.638,Z 398.858,A -85,B 0,C 180,E1 -7233.221,E2 -7233.221} C_VEL
LIN {X 0,Y 474.589,Z 398.87,A -85,B 0,C 180,E1 -7236.324,E2 -7236.324} C_VEL
LIN {X 0,Y 474.646,Z 398.864,A -85,B 0,C 180,E1 -7239.652,E2 -7239.652} C_VEL
LIN {X 0,Y 474.626,Z 399.004,A -85,B 0,C 180,E1 -7242.238,E2 -7242.238} C_VEL
LIN {X 0,Y 475.114,Z 402.477,A -85,B 0,C 180,E1 -7245.238,E2 -7245.238} C_VEL
LIN {X 0,Y 475.432,Z 405.534,A -85,B 0,C 180,E1 -7247.657,E2 -7247.657} C_VEL
LIN {X 0,Y 475.338,Z 409.082,A -85,B 0,C 180,E1 -7250.25,E2 -7250.25} C_VEL
LIN {X 0,Y 475.173,Z 413.106,A -85,B 0,C 180,E1 -7253.005,E2 -7253.005} C_VEL
LIN {X 0,Y 474.93,Z 417.69,A -85,B 0,C 180,E1 -7255.965,E2 -7255.965} C_VEL
LIN {X 0,Y 474.689,Z 422.324,A -85,B 0,C 180,E1 -7258.79,E2 -7258.79} C_VEL
LIN {X 0,Y 474.473,Z 427.308,A -85,B 0,C 180,E1 -7261.707,E2 -7261.707} C_VEL
LIN {X 0,Y 474.267,Z 432.618,A -85,B 0,C 180,E1 -7264.681,E2 -7264.681} C_VEL
LIN {X 0,Y 474.11,Z 437.524,A -85,B 0,C 180,E1 -7267.331,E2 -7267.331} C_VEL
LIN {X 0,Y 474.101,Z 440.97,A -85,B 0,C 180,E1 -7269.16,E2 -7269.16} C_VEL
LIN {X 0,Y 473.941,Z 446.185,A -85,B 0,C 180,E1 -7271.856,E2 -7271.856} C_VEL
LIN {X 0,Y 473.911,Z 452.235,A -85,B 0,C 180,E1 -7274.866,E2 -7274.866} C_VEL
LIN {X 0,Y 475.576,Z 462.498,A -85,B 0,C 180,E1 -7275.185,E2 -7275.185} C_VEL
LIN {X 0,Y 476.859,Z 471.369,A -85,B 0,C 180,E1 -7275.545,E2 -7275.545} C_VEL
LIN {X 0,Y 476.616,Z 480.728,A -85,B 0,C 180,E1 -7275.973,E2 -7275.973} C_VEL
LIN {X 0,Y 476.188,Z 491.197,A -85,B 0,C 180,E1 -7276.581,E2 -7276.581} C_VEL
LIN {X 0,Y 475.808,Z 499.869,A -85,B 0,C 180,E1 -7277.2,E2 -7277.2} C_VEL
LIN {X 0,Y 475.487,Z 508.664,A -85,B 0,C 180,E1 -7277.956,E2 -7277.956} C_VEL
LIN {X 0,Y 475.15,Z 515.999,A -85,B 0,C 180,E1 -7278.698,E2 -7278.698} C_VEL
LIN {X 0,Y 474.779,Z 523.219,A -85,B 0,C 180,E1 -7279.553,E2 -7279.553} C_VEL
LIN {X 0,Y 474.495,Z 529.422,A -85,B 0,C 180,E1 -7280.408,E2 -7280.408} C_VEL
LIN {X 0,Y 474.27,Z 535.961,A -85,B 0,C 180,E1 -7281.478,E2 -7281.478} C_VEL
LIN {X 0,Y 474.065,Z 540.461,A -85,B 0,C 180,E1 -7282.333,E2 -7282.333} C_VEL
LIN {X 0,Y 473.881,Z 545.707,A -85,B 0,C 180,E1 -7283.547,E2 -7283.547} C_VEL
LIN {X 0,Y 473.836,Z 550.274,A -85,B 0,C 180,E1 -7284.894,E2 -7284.894} C_VEL
LIN {X 0,Y 473.742,Z 552.637,A -85,B 0,C 180,E1 -7285.746,E2 -7285.746} C_VEL
LIN {X 0,Y 473.797,Z 554.435,A -85,B 0,C 180,E1 -7286.599,E2 -7286.599} C_VEL
LIN {X 0,Y 473.698,Z 556.874,A -85,B 0,C 180,E1 -7288.3,E2 -7288.3} C_VEL
LIN {X 0,Y 473.688,Z 557.461,A -85,B 0,C 180,E1 -7289.15,E2 -7289.15} C_VEL
LIN {X 0,Y 473.688,Z 557.461,A -85,B 0,C 180,E1 -7290.85,E2 -7290.85} C_VEL
LIN {X 0,Y 473.698,Z 556.874,A -85,B 0,C 180,E1 -7291.7,E2 -7291.7} C_VEL
LIN {X 0,Y 473.797,Z 554.435,A -85,B 0,C 180,E1 -7293.401,E2 -7293.401} C_VEL
LIN {X 0,Y 473.771,Z 551.488,A -85,B 0,C 180,E1 -7294.68,E2 -7294.68} C_VEL
LIN {X 0,Y 473.852,Z 547.504,A -85,B 0,C 180,E1 -7295.959,E2 -7295.959} C_VEL
LIN {X 0,Y 474.012,Z 542.377,A -85,B 0,C 180,E1 -7297.24,E2 -7297.24} C_VEL
LIN {X 0,Y 474.195,Z 537.115,A -85,B 0,C 180,E1 -7298.308,E2 -7298.308} C_VEL
LIN {X 0,Y 474.424,Z 530.798,A -85,B 0,C 180,E1 -7299.378,E2 -7299.378} C_VEL
LIN {X 0,Y 474.678,Z 524.845,A -85,B 0,C 180,E1 -7300.234,E2 -7300.234} C_VEL
LIN {X 0,Y 475.042,Z 517.918,A -85,B 0,C 180,E1 -7301.088,E2 -7301.088} C_VEL
LIN {X 0,Y 475.451,Z 509.737,A -85,B 0,C 180,E1 -7301.943,E2 -7301.943} C_VEL
LIN {X 0,Y 475.724,Z 501.864,A -85,B 0,C 180,E1 -7302.643,E2 -7302.643} C_VEL
LIN {X 0,Y 476.09,Z 492.992,A -85,B 0,C 180,E1 -7303.303,E2 -7303.303} C_VEL
LIN {X 0,Y 476.52,Z 482.742,A -85,B 0,C 180,E1 -7303.921,E2 -7303.921} C_VEL
LIN {X 0,Y 476.864,Z 472.659,A -85,B 0,C 180,E1 -7304.4,E2 -7304.4} C_VEL
LIN {X 0,Y 475.723,Z 463.349,A -85,B 0,C 180,E1 -7304.783,E2 -7304.783} C_VEL
LIN {X 0,Y 474.009,Z 453.205,A -85,B 0,C 180,E1 -7305.111,E2 -7305.111} C_VEL
LIN {X 0,Y 473.888,Z 452.109,A -85,B 0,C 180,E1 -7305.162,E2 -7305.162} C_VEL
LIN {X 0,Y 473.949,Z 445.736,A -85,B 0,C 180,E1 -7308.371,E2 -7308.371} C_VEL
LIN {X 0,Y 474.081,Z 440.772,A -85,B 0,C 180,E1 -7310.941,E2 -7310.941} C_VEL
LIN {X 0,Y 474.153,Z 435.789,A -85,B 0,C 180,E1 -7313.59,E2 -7313.59} C_VEL
LIN {X 0,Y 474.347,Z 430.674,A -85,B 0,C 180,E1 -7316.39,E2 -7316.39} C_VEL
LIN {X 0,Y 474.538,Z 425.626,A -85,B 0,C 180,E1 -7319.257,E2 -7319.257} C_VEL
LIN {X 0,Y 474.816,Z 420.207,A -85,B 0,C 180,E1 -7322.468,E2 -7322.468} C_VEL
LIN {X 0,Y 475.07,Z 415.304,A -85,B 0,C 180,E1 -7325.546,E2 -7325.546} C_VEL
LIN {X 0,Y 475.259,Z 411.014,A -85,B 0,C 180,E1 -7328.394,E2 -7328.394} C_VEL
LIN {X 0,Y 475.444,Z 406.378,A -85,B 0,C 180,E1 -7331.696,E2 -7331.696} C_VEL
LIN {X 0,Y 475.245,Z 403.362,A -85,B 0,C 180,E1 -7334.029,E2 -7334.029} C_VEL
LIN {X 0,Y 474.741,Z 399.767,A -85,B 0,C 180,E1 -7337.079,E2 -7337.079} C_VEL
LIN {X 0,Y 474.626,Z 399.003,A -85,B 0,C 180,E1 -7337.762,E2 -7337.762} C_VEL
LIN {X 0,Y 474.664,Z 398.861,A -85,B 0,C 180,E1 -7340.456,E2 -7340.456} C_VEL
LIN {X 0,Y 474.589,Z 398.87,A -85,B 0,C 180,E1 -7343.676,E2 -7343.676} C_VEL
LIN {X 0,Y 474.638,Z 398.858,A -85,B 0,C 180,E1 -7346.779,E2 -7346.779} C_VEL
LIN {X 0,Y 474.609,Z 398.867,A -85,B 0,C 180,E1 -7349.77,E2 -7349.77} C_VEL
LIN {X 0,Y 474.691,Z 398.851,A -85,B 0,C 180,E1 -7352.679,E2 -7352.679} C_VEL
LIN {X 0,Y 474.652,Z 398.859,A -85,B 0,C 180,E1 -7355.506,E2 -7355.506} C_VEL
LIN {X 0,Y 474.663,Z 398.855,A -85,B 0,C 180,E1 -7359.185,E2 -7359.185} C_VEL
LIN {X 0,Y 474.65,Z 398.863,A -85,B 0,C 180,E1 -7361.884,E2 -7361.884} C_VEL
LIN {X 0,Y 474.692,Z 398.851,A -85,B 0,C 180,E1 -7364.544,E2 -7364.544} C_VEL
LIN {X 0,Y 474.696,Z 398.853,A -85,B 0,C 180,E1 -7368.037,E2 -7368.037} C_VEL
LIN {X 0,Y 474.72,Z 398.854,A -85,B 0,C 180,E1 -7371.486,E2 -7371.486} C_VEL
LIN {X 0,Y 474.771,Z 398.843,A -85,B 0,C 180,E1 -7374.052,E2 -7374.052} C_VEL
LIN {X 0,Y 474.886,Z 398.834,A -85,B 0,C 180,E1 -7377.455,E2 -7377.455} C_VEL
LIN {X 0,Y 474.902,Z 398.826,A -85,B 0,C 180,E1 -7380,E2 -7380} C_VEL
LIN {X 0,Y 474.886,Z 398.826,A -85,B 0,C 180,E1 -7382.544,E2 -7382.544} C_VEL
LIN {X 0,Y 474.774,Z 398.842,A -85,B 0,C 180,E1 -7385.947,E2 -7385.947} C_VEL
LIN {X 0,Y 474.719,Z 398.847,A -85,B 0,C 180,E1 -7388.513,E2 -7388.513} C_VEL
LIN {X 0,Y 474.694,Z 398.851,A -85,B 0,C 180,E1 -7391.962,E2 -7391.962} C_VEL
LIN {X 0,Y 474.69,Z 398.856,A -85,B 0,C 180,E1 -7395.455,E2 -7395.455} C_VEL
LIN {X 0,Y 474.656,Z 398.861,A -85,B 0,C 180,E1 -7399.01,E2 -7399.01} C_VEL
LIN {X 0,Y 474.579,Z 398.866,A -85,B 0,C 180,E1 -7401.729,E2 -7401.729} C_VEL
LIN {X 0,Y 474.649,Z 398.857,A -85,B 0,C 180,E1 -7404.493,E2 -7404.493} C_VEL
LIN {X 0,Y 474.69,Z 398.855,A -85,B 0,C 180,E1 -7407.339,E2 -7407.339} C_VEL
LIN {X 0,Y 474.601,Z 398.868,A -85,B 0,C 180,E1 -7410.811,E2 -7410.811} C_VEL
LIN {X 0,Y 474.629,Z 398.858,A -85,B 0,C 180,E1 -7413.984,E2 -7413.984} C_VEL
LIN {X 0,Y 474.568,Z 398.874,A -85,B 0,C 180,E1 -7416.9,E2 -7416.9} C_VEL
LIN {X 0,Y 474.646,Z 398.856,A -85,B 0,C 180,E1 -7419.652,E2 -7419.652} C_VEL
LIN {X 0,Y 474.644,Z 398.863,A -85,B 0,C 180,E1 -7422.93,E2 -7422.93} C_VEL
LIN {X 0,Y 474.607,Z 398.861,A -85,B 0,C 180,E1 -7425.896,E2 -7425.896} C_VEL
LIN {X 0,Y 474.625,Z 398.862,A -85,B 0,C 180,E1 -7429.04,E2 -7429.04} C_VEL
LIN {X 0,Y 474.603,Z 398.862,A -85,B 0,C 180,E1 -7431.704,E2 -7431.704} C_VEL
LIN {X 0,Y 474.624,Z 398.865,A -85,B 0,C 180,E1 -7434.727,E2 -7434.727} C_VEL
LIN {X 0,Y 474.631,Z 398.859,A -85,B 0,C 180,E1 -7437.788,E2 -7437.788} C_VEL
LIN {X 0,Y 474.618,Z 398.863,A -85,B 0,C 180,E1 -7440.885,E2 -7440.885} C_VEL
LIN {X 0,Y 474.661,Z 398.855,A -85,B 0,C 180,E1 -7443.629,E2 -7443.629} C_VEL
LIN {X 0,Y 474.631,Z 398.863,A -85,B 0,C 180,E1 -7446.641,E2 -7446.641} C_VEL
LIN {X 0,Y 474.65,Z 398.861,A -85,B 0,C 180,E1 -7450.09,E2 -7450.09} C_VEL
LIN {X 0,Y 474.651,Z 398.86,A -85,B 0,C 180,E1 -7451.68,E2 -7451.68} C_VEL
LIN {X 0,Y 473.988,Z 398.946,A -85,B 0,C 180,E1 -7452.389,E2 -7452.389} C_VEL
LIN {X 0,Y 471.137,Z 399.3,A -85,B 0,C 180,E1 -7453.541,E2 -7453.541} C_VEL
LIN {X 0,Y 468.721,Z 399.602,A -85,B 0,C 180,E1 -7454.469,E2 -7454.469} C_VEL
LIN {X 0,Y 467.679,Z 399.727,A -85,B 0,C 180,E1 -7455.186,E2 -7455.186} C_VEL
LIN {X 0,Y 467.592,Z 399.738,A -85,B 0,C 180,E1 -7455.429,E2 -7455.429} C_VEL
LIN {X 0,Y 467.65,Z 399.733,A -85,B 0,C 180,E1 -7458.734,E2 -7458.734} C_VEL
LIN {X 0,Y 467.745,Z 399.724,A -85,B 0,C 180,E1 -7462.228,E2 -7462.228} C_VEL
LIN {X 0,Y 467.722,Z 399.723,A -85,B 0,C 180,E1 -7464.828,E2 -7464.828} C_VEL
LIN {X 0,Y 467.857,Z 399.706,A -85,B 0,C 180,E1 -7467.417,E2 -7467.417} C_VEL
LIN {X 0,Y 467.88,Z 399.708,A -85,B 0,C 180,E1 -7470,E2 -7470} C_VEL
LIN {X 0,Y 467.857,Z 399.706,A -85,B 0,C 180,E1 -7472.583,E2 -7472.583} C_VEL
LIN {X 0,Y 467.741,Z 399.724,A -85,B 0,C 180,E1 -7476.037,E2 -7476.037} C_VEL
LIN {X 0,Y 467.678,Z 399.729,A -85,B 0,C 180,E1 -7478.643,E2 -7478.643} C_VEL
LIN {X 0,Y 467.652,Z 399.734,A -85,B 0,C 180,E1 -7482.145,E2 -7482.145} C_VEL
LIN {X 0,Y 467.635,Z 399.738,A -85,B 0,C 180,E1 -7485.695,E2 -7485.695} C_VEL
LIN {X 0,Y 467.613,Z 399.735,A -85,B 0,C 180,E1 -7488.764,E2 -7488.764} C_VEL
LIN {X 0,Y 467.576,Z 399.74,A -85,B 0,C 180,E1 -7491.268,E2 -7491.268} C_VEL
LIN {X 0,Y 467.568,Z 399.742,A -85,B 0,C 180,E1 -7493.943,E2 -7493.943} C_VEL
LIN {X 0,Y 467.622,Z 399.732,A -85,B 0,C 180,E1 -7496.799,E2 -7496.799} C_VEL
LIN {X 0,Y 467.548,Z 399.746,A -85,B 0,C 180,E1 -7499.738,E2 -7499.738} C_VEL
LIN {X 0,Y 467.577,Z 399.738,A -85,B 0,C 180,E1 -7502.758,E2 -7502.758} C_VEL
LIN {X 0,Y 467.55,Z 399.743,A -85,B 0,C 180,E1 -7505.889,E2 -7505.889} C_VEL
LIN {X 0,Y 467.575,Z 399.742,A -85,B 0,C 180,E1 -7509.144,E2 -7509.144} C_VEL
LIN {X 0,Y 467.579,Z 399.737,A -85,B 0,C 180,E1 -7512.567,E2 -7512.567} C_VEL
LIN {X 0,Y 467.563,Z 399.744,A -85,B 0,C 180,E1 -7515.053,E2 -7515.053} C_VEL
LIN {X 0,Y 467.58,Z 399.742,A -85,B 0,C 180,E1 -7517.44,E2 -7517.44} C_VEL
LIN {X 0,Y 467.574,Z 399.741,A -85,B 0,C 180,E1 -7520.855,E2 -7520.855} C_VEL
LIN {X 0,Y 467.554,Z 399.74,A -85,B 0,C 180,E1 -7524.26,E2 -7524.26} C_VEL
LIN {X 0,Y 467.573,Z 399.742,A -85,B 0,C 180,E1 -7527.321,E2 -7527.321} C_VEL
LIN {X 0,Y 467.569,Z 399.742,A -85,B 0,C 180,E1 -7530.665,E2 -7530.665} C_VEL
LIN {X 0,Y 467.618,Z 399.737,A -85,B 0,C 180,E1 -7533.2,E2 -7533.2} C_VEL
LIN {X 0,Y 467.583,Z 399.739,A -85,B 0,C 180,E1 -7536.468,E2 -7536.468} C_VEL
LIN {X 0,Y 467.614,Z 399.732,A -85,B 0,C 180,E1 -7539.777,E2 -7539.777} C_VEL
LIN {X 0,Y 467.6,Z 399.738,A -85,B 0,C 180,E1 -7542.507,E2 -7542.507} C_VEL
LIN {X 0,Y 467.597,Z 399.737,A -85,B 0,C 180,E1 -7545.197,E2 -7545.197} C_VEL
LIN {X 0,Y 467.646,Z 399.728,A -85,B 0,C 180,E1 -7547.855,E2 -7547.855} C_VEL
LIN {X 0,Y 467.672,Z 399.726,A -85,B 0,C 180,E1 -7551.358,E2 -7551.358} C_VEL
LIN {X 0,Y 467.738,Z 399.718,A -85,B 0,C 180,E1 -7553.963,E2 -7553.963} C_VEL
LIN {X 0,Y 467.852,Z 399.703,A -85,B 0,C 180,E1 -7557.418,E2 -7557.418} C_VEL
LIN {X 0,Y 467.873,Z 399.702,A -85,B 0,C 180,E1 -7560,E2 -7560} C_VEL
LIN {X 0,Y 467.852,Z 399.71,A -85,B 0,C 180,E1 -7562.583,E2 -7562.583} C_VEL
LIN {X 0,Y 467.735,Z 399.72,A -85,B 0,C 180,E1 -7566.038,E2 -7566.038} C_VEL
LIN {X 0,Y 467.674,Z 399.73,A -85,B 0,C 180,E1 -7568.643,E2 -7568.643} C_VEL
LIN {X 0,Y 467.647,Z 399.734,A -85,B 0,C 180,E1 -7572.146,E2 -7572.146} C_VEL
LIN {X 0,Y 467.659,Z 399.73,A -85,B 0,C 180,E1 -7575.893,E2 -7575.893} C_VEL
LIN {X 0,Y 467.616,Z 399.732,A -85,B 0,C 180,E1 -7579.309,E2 -7579.309} C_VEL
LIN {X 0,Y 467.528,Z 399.75,A -85,B 0,C 180,E1 -7582.075,E2 -7582.075} C_VEL
LIN {X 0,Y 467.597,Z 399.735,A -85,B 0,C 180,E1 -7584.888,E2 -7584.888} C_VEL
LIN {X 0,Y 467.615,Z 399.736,A -85,B 0,C 180,E1 -7587.77,E2 -7587.77} C_VEL
LIN {X 0,Y 467.567,Z 399.738,A -85,B 0,C 180,E1 -7591.047,E2 -7591.047} C_VEL
LIN {X 0,Y 467.586,Z 399.743,A -85,B 0,C 180,E1 -7594.244,E2 -7594.244} C_VEL
LIN {X 0,Y 467.546,Z 399.745,A -85,B 0,C 180,E1 -7597.188,E2 -7597.188} C_VEL
LIN {X 0,Y 467.591,Z 399.743,A -85,B 0,C 180,E1 -7600.264,E2 -7600.264} C_VEL
LIN {X 0,Y 467.577,Z 399.745,A -85,B 0,C 180,E1 -7601.403,E2 -7601.403} C_VEL
LIN {X 0,Y 467.679,Z 400.59,A -85,B 0,C 180,E1 -7602.581,E2 -7602.581} C_VEL
LIN {X 0,Y 468.121,Z 403.502,A -85,B 0,C 180,E1 -7605.122,E2 -7605.122} C_VEL
LIN {X 0,Y 468.409,Z 406.477,A -85,B 0,C 180,E1 -7607.533,E2 -7607.533} C_VEL
LIN {X 0,Y 468.325,Z 409.697,A -85,B 0,C 180,E1 -7609.938,E2 -7609.938} C_VEL
LIN {X 0,Y 468.122,Z 414.239,A -85,B 0,C 180,E1 -7613.093,E2 -7613.093} C_VEL
LIN {X 0,Y 467.848,Z 419.036,A -85,B 0,C 180,E1 -7616.234,E2 -7616.234} C_VEL
LIN {X 0,Y 467.625,Z 423.958,A -85,B 0,C 180,E1 -7619.271,E2 -7619.271} C_VEL
LIN {X 0,Y 467.381,Z 429.473,A -85,B 0,C 180,E1 -7622.522,E2 -7622.522} C_VEL
LIN {X 0,Y 467.168,Z 434.007,A -85,B 0,C 180,E1 -7625.088,E2 -7625.088} C_VEL
LIN {X 0,Y 466.992,Z 439.145,A -85,B 0,C 180,E1 -7627.9,E2 -7627.9} C_VEL
LIN {X 0,Y 466.865,Z 444.334,A -85,B 0,C 180,E1 -7630.66,E2 -7630.66} C_VEL
LIN {X 0,Y 466.778,Z 449.544,A -85,B 0,C 180,E1 -7633.377,E2 -7633.377} C_VEL
LIN {X 0,Y 466.813,Z 452.119,A -85,B 0,C 180,E1 -7634.632,E2 -7634.632} C_VEL
LIN {X 0,Y 468.537,Z 462.324,A -85,B 0,C 180,E1 -7634.959,E2 -7634.959} C_VEL
LIN {X 0,Y 469.965,Z 472.461,A -85,B 0,C 180,E1 -7635.383,E2 -7635.383} C_VEL
LIN {X 0,Y 469.639,Z 482.545,A -85,B 0,C 180,E1 -7635.871,E2 -7635.871} C_VEL
LIN {X 0,Y 469.203,Z 492.31,A -85,B 0,C 180,E1 -7636.466,E2 -7636.466} C_VEL
LIN {X 0,Y 468.762,Z 502.083,A -85,B 0,C 180,E1 -7637.2,E2 -7637.2} C_VEL
LIN {X 0,Y 468.299,Z 512.898,A -85,B 0,C 180,E1 -7638.201,E2 -7638.201} C_VEL
LIN {X 0,Y 467.835,Z 521.393,A -85,B 0,C 180,E1 -7639.177,E2 -7639.177} C_VEL
LIN {X 0,Y 467.478,Z 529.224,A -85,B 0,C 180,E1 -7640.263,E2 -7640.263} C_VEL
LIN {X 0,Y 467.208,Z 535.762,A -85,B 0,C 180,E1 -7641.349,E2 -7641.349} C_VEL
LIN {X 0,Y 467.01,Z 540.263,A -85,B 0,C 180,E1 -7642.216,E2 -7642.216} C_VEL
LIN {X 0,Y 466.808,Z 545.862,A -85,B 0,C 180,E1 -7643.547,E2 -7643.547} C_VEL
LIN {X 0,Y 466.746,Z 550.076,A -85,B 0,C 180,E1 -7644.817,E2 -7644.817} C_VEL
LIN {X 0,Y 466.654,Z 552.439,A -85,B 0,C 180,E1 -7645.682,E2 -7645.682} C_VEL
LIN {X 0,Y 466.692,Z 554.237,A -85,B 0,C 180,E1 -7646.547,E2 -7646.547} C_VEL
LIN {X 0,Y 466.608,Z 556.677,A -85,B 0,C 180,E1 -7648.274,E2 -7648.274} C_VEL
LIN {X 0,Y 466.619,Z 557.265,A -85,B 0,C 180,E1 -7649.137,E2 -7649.137} C_VEL
LIN {X 0,Y 466.619,Z 557.265,A -85,B 0,C 180,E1 -7650.863,E2 -7650.863} C_VEL
LIN {X 0,Y 466.608,Z 556.677,A -85,B 0,C 180,E1 -7651.726,E2 -7651.726} C_VEL
LIN {X 0,Y 466.692,Z 554.237,A -85,B 0,C 180,E1 -7653.453,E2 -7653.453} C_VEL
LIN {X 0,Y 466.698,Z 551.291,A -85,B 0,C 180,E1 -7654.751,E2 -7654.751} C_VEL
LIN {X 0,Y 466.767,Z 547.306,A -85,B 0,C 180,E1 -7656.05,E2 -7656.05} C_VEL
LIN {X 0,Y 466.943,Z 542.179,A -85,B 0,C 180,E1 -7657.35,E2 -7657.35} C_VEL
LIN {X 0,Y 467.155,Z 536.918,A -85,B 0,C 180,E1 -7658.434,E2 -7658.434} C_VEL
LIN {X 0,Y 467.393,Z 530.6,A -85,B 0,C 180,E1 -7659.52,E2 -7659.52} C_VEL
LIN {X 0,Y 467.654,Z 524.647,A -85,B 0,C 180,E1 -7660.389,E2 -7660.389} C_VEL
LIN {X 0,Y 468.039,Z 517.72,A -85,B 0,C 180,E1 -7661.256,E2 -7661.256} C_VEL
LIN {X 0,Y 468.479,Z 509.54,A -85,B 0,C 180,E1 -7662.123,E2 -7662.123} C_VEL
LIN {X 0,Y 468.745,Z 501.665,A -85,B 0,C 180,E1 -7662.834,E2 -7662.834} C_VEL
LIN {X 0,Y 469.204,Z 492.305,A -85,B 0,C 180,E1 -7663.535,E2 -7663.535} C_VEL
LIN {X 0,Y 469.631,Z 482.545,A -85,B 0,C 180,E1 -7664.129,E2 -7664.129} C_VEL
LIN {X 0,Y 469.993,Z 472.462,A -85,B 0,C 180,E1 -7664.616,E2 -7664.616} C_VEL
LIN {X 0,Y 468.521,Z 461.973,A -85,B 0,C 180,E1 -7665.053,E2 -7665.053} C_VEL
LIN {X 0,Y 466.82,Z 451.944,A -85,B 0,C 180,E1 -7665.398,E2 -7665.398} C_VEL
LIN {X 0,Y 466.879,Z 445.917,A -85,B 0,C 180,E1 -7668.494,E2 -7668.494} C_VEL
LIN {X 0,Y 466.992,Z 440.853,A -85,B 0,C 180,E1 -7671.173,E2 -7671.173} C_VEL
LIN {X 0,Y 467.107,Z 435.704,A -85,B 0,C 180,E1 -7673.968,E2 -7673.968} C_VEL
LIN {X 0,Y 467.299,Z 430.619,A -85,B 0,C 180,E1 -7676.819,E2 -7676.819} C_VEL
LIN {X 0,Y 467.5,Z 425.596,A -85,B 0,C 180,E1 -7679.741,E2 -7679.741} C_VEL
LIN {X 0,Y 467.78,Z 420.656,A -85,B 0,C 180,E1 -7682.742,E2 -7682.742} C_VEL
LIN {X 0,Y 468.043,Z 415.812,A -85,B 0,C 180,E1 -7685.845,E2 -7685.845} C_VEL
LIN {X 0,Y 468.235,Z 411.62,A -85,B 0,C 180,E1 -7688.693,E2 -7688.693} C_VEL
LIN {X 0,Y 468.415,Z 407.865,A -85,B 0,C 180,E1 -7691.393,E2 -7691.393} C_VEL
LIN {X 0,Y 468.281,Z 404.632,A -85,B 0,C 180,E1 -7693.913,E2 -7693.913} C_VEL
LIN {X 0,Y 467.687,Z 400.552,A -85,B 0,C 180,E1 -7697.45,E2 -7697.45} C_VEL
LIN {X 0,Y 467.58,Z 399.743,A -85,B 0,C 180,E1 -7698.721,E2 -7698.721} C_VEL
LIN {X 0,Y 467.57,Z 399.743,A -85,B 0,C 180,E1 -7701.406,E2 -7701.406} C_VEL
LIN {X 0,Y 467.559,Z 399.748,A -85,B 0,C 180,E1 -7704.259,E2 -7704.259} C_VEL
LIN {X 0,Y 467.577,Z 399.738,A -85,B 0,C 180,E1 -7707.32,E2 -7707.32} C_VEL
LIN {X 0,Y 467.572,Z 399.738,A -85,B 0,C 180,E1 -7710.665,E2 -7710.665} C_VEL
LIN {X 0,Y 467.61,Z 399.734,A -85,B 0,C 180,E1 -7713.199,E2 -7713.199} C_VEL
LIN {X 0,Y 467.586,Z 399.737,A -85,B 0,C 180,E1 -7716.467,E2 -7716.467} C_VEL
LIN {X 0,Y 467.615,Z 399.74,A -85,B 0,C 180,E1 -7719.776,E2 -7719.776} C_VEL
LIN {X 0,Y 467.602,Z 399.734,A -85,B 0,C 180,E1 -7722.506,E2 -7722.506} C_VEL
LIN {X 0,Y 467.599,Z 399.736,A -85,B 0,C 180,E1 -7725.196,E2 -7725.196} C_VEL
LIN {X 0,Y 467.647,Z 399.734,A -85,B 0,C 180,E1 -7727.854,E2 -7727.854} C_VEL
LIN {X 0,Y 467.674,Z 399.73,A -85,B 0,C 180,E1 -7731.357,E2 -7731.357} C_VEL
LIN {X 0,Y 467.735,Z 399.72,A -85,B 0,C 180,E1 -7733.962,E2 -7733.962} C_VEL
LIN {X 0,Y 467.852,Z 399.71,A -85,B 0,C 180,E1 -7737.417,E2 -7737.417} C_VEL
LIN {X 0,Y 467.873,Z 399.702,A -85,B 0,C 180,E1 -7740,E2 -7740} C_VEL
LIN {X 0,Y 467.852,Z 399.703,A -85,B 0,C 180,E1 -7742.582,E2 -7742.582} C_VEL
LIN {X 0,Y 467.738,Z 399.718,A -85,B 0,C 180,E1 -7746.037,E2 -7746.037} C_VEL
LIN {X 0,Y 467.673,Z 399.726,A -85,B 0,C 180,E1 -7748.642,E2 -7748.642} C_VEL
LIN {X 0,Y 467.646,Z 399.728,A -85,B 0,C 180,E1 -7752.145,E2 -7752.145} C_VEL
LIN {X 0,Y 467.629,Z 399.733,A -85,B 0,C 180,E1 -7755.695,E2 -7755.695} C_VEL
LIN {X 0,Y 467.608,Z 399.736,A -85,B 0,C 180,E1 -7758.765,E2 -7758.765} C_VEL
LIN {X 0,Y 467.57,Z 399.744,A -85,B 0,C 180,E1 -7761.268,E2 -7761.268} C_VEL
LIN {X 0,Y 467.563,Z 399.739,A -85,B 0,C 180,E1 -7763.943,E2 -7763.943} C_VEL
LIN {X 0,Y 467.618,Z 399.737,A -85,B 0,C 180,E1 -7766.8,E2 -7766.8} C_VEL
LIN {X 0,Y 467.578,Z 399.737,A -85,B 0,C 180,E1 -7769.736,E2 -7769.736} C_VEL
LIN {X 0,Y 467.575,Z 399.743,A -85,B 0,C 180,E1 -7772.758,E2 -7772.758} C_VEL
LIN {X 0,Y 467.548,Z 399.741,A -85,B 0,C 180,E1 -7775.889,E2 -7775.889} C_VEL
LIN {X 0,Y 467.61,Z 399.737,A -85,B 0,C 180,E1 -7779.141,E2 -7779.141} C_VEL
LIN {X 0,Y 467.611,Z 399.738,A -85,B 0,C 180,E1 -7782.572,E2 -7782.572} C_VEL
LIN {X 0,Y 467.559,Z 399.741,A -85,B 0,C 180,E1 -7786.178,E2 -7786.178} C_VEL
LIN {X 0,Y 467.574,Z 399.745,A -85,B 0,C 180,E1 -7788.723,E2 -7788.723} C_VEL
LIN {X 0,Y 467.559,Z 399.74,A -85,B 0,C 180,E1 -7791.956,E2 -7791.956} C_VEL
LIN {X 0,Y 467.562,Z 399.74,A -85,B 0,C 180,E1 -7795.168,E2 -7795.168} C_VEL
LIN {X 0,Y 467.578,Z 399.741,A -85,B 0,C 180,E1 -7798.26,E2 -7798.26} C_VEL
LIN {X 0,Y 467.571,Z 399.738,A -85,B 0,C 180,E1 -7801.251,E2 -7801.251} C_VEL
LIN {X 0,Y 467.607,Z 399.738,A -85,B 0,C 180,E1 -7804.16,E2 -7804.16} C_VEL
LIN {X 0,Y 467.573,Z 399.739,A -85,B 0,C 180,E1 -7806.996,E2 -7806.996} C_VEL
LIN {X 0,Y 467.618,Z 399.733,A -85,B 0,C 180,E1 -7809.777,E2 -7809.777} C_VEL
LIN {X 0,Y 467.604,Z 399.74,A -85,B 0,C 180,E1 -7812.507,E2 -7812.507} C_VEL
LIN {X 0,Y 467.592,Z 399.738,A -85,B 0,C 180,E1 -7815.429,E2 -7815.429} C_VEL
LIN {X 0,Y 466.923,Z 399.827,A -85,B 0,C 180,E1 -7816.149,E2 -7816.149} C_VEL
LIN {X 0,Y 464.079,Z 400.177,A -85,B 0,C 180,E1 -7817.317,E2 -7817.317} C_VEL
LIN {X 0,Y 461.681,Z 400.478,A -85,B 0,C 180,E1 -7818.259,E2 -7818.259} C_VEL
LIN {X 0,Y 460.655,Z 400.603,A -85,B 0,C 180,E1 -7818.987,E2 -7818.987} C_VEL
LIN {X 0,Y 460.574,Z 400.613,A -85,B 0,C 180,E1 -7819.233,E2 -7819.233} C_VEL
LIN {X 0,Y 460.716,Z 400.597,A -85,B 0,C 180,E1 -7822.538,E2 -7822.538} C_VEL
LIN {X 0,Y 460.695,Z 400.599,A -85,B 0,C 180,E1 -7824.748,E2 -7824.748} C_VEL
LIN {X 0,Y 460.822,Z 400.583,A -85,B 0,C 180,E1 -7827.378,E2 -7827.378} C_VEL
LIN {X 0,Y 460.85,Z 400.583,A -85,B 0,C 180,E1 -7830,E2 -7830} C_VEL
LIN {X 0,Y 460.822,Z 400.583,A -85,B 0,C 180,E1 -7832.622,E2 -7832.622} C_VEL
LIN {X 0,Y 460.707,Z 400.6,A -85,B 0,C 180,E1 -7836.13,E2 -7836.13} C_VEL
LIN {X 0,Y 460.625,Z 400.607,A -85,B 0,C 180,E1 -7838.776,E2 -7838.776} C_VEL
LIN {X 0,Y 460.609,Z 400.609,A -85,B 0,C 180,E1 -7842.445,E2 -7842.445} C_VEL
LIN {X 0,Y 460.596,Z 400.614,A -85,B 0,C 180,E1 -7845.997,E2 -7845.997} C_VEL
LIN {X 0,Y 460.566,Z 400.614,A -85,B 0,C 180,E1 -7848.902,E2 -7848.902} C_VEL
LIN {X 0,Y 460.511,Z 400.623,A -85,B 0,C 180,E1 -7851.485,E2 -7851.485} C_VEL
LIN {X 0,Y 460.537,Z 400.614,A -85,B 0,C 180,E1 -7854.332,E2 -7854.332} C_VEL
LIN {X 0,Y 460.578,Z 400.613,A -85,B 0,C 180,E1 -7857.243,E2 -7857.243} C_VEL
LIN {X 0,Y 460.505,Z 400.618,A -85,B 0,C 180,E1 -7860.24,E2 -7860.24} C_VEL
LIN {X 0,Y 460.523,Z 400.622,A -85,B 0,C 180,E1 -7863.324,E2 -7863.324} C_VEL
LIN {X 0,Y 460.472,Z 400.622,A -85,B 0,C 180,E1 -7866.529,E2 -7866.529} C_VEL
LIN {X 0,Y 460.551,Z 400.614,A -85,B 0,C 180,E1 -7869.859,E2 -7869.859} C_VEL
LIN {X 0,Y 460.509,Z 400.62,A -85,B 0,C 180,E1 -7872.901,E2 -7872.901} C_VEL
LIN {X 0,Y 460.512,Z 400.619,A -85,B 0,C 180,E1 -7875.829,E2 -7875.829} C_VEL
LIN {X 0,Y 460.525,Z 400.621,A -85,B 0,C 180,E1 -7878.989,E2 -7878.989} C_VEL
LIN {X 0,Y 460.518,Z 400.623,A -85,B 0,C 180,E1 -7881.267,E2 -7881.267} C_VEL
LIN {X 0,Y 460.505,Z 400.62,A -85,B 0,C 180,E1 -7884.555,E2 -7884.555} C_VEL
LIN {X 0,Y 460.523,Z 400.617,A -85,B 0,C 180,E1 -7887.716,E2 -7887.716} C_VEL
LIN {X 0,Y 460.538,Z 400.619,A -85,B 0,C 180,E1 -7890.77,E2 -7890.77} C_VEL
LIN {X 0,Y 460.559,Z 400.612,A -85,B 0,C 180,E1 -7893.735,E2 -7893.735} C_VEL
LIN {X 0,Y 460.536,Z 400.618,A -85,B 0,C 180,E1 -7896.624,E2 -7896.624} C_VEL
LIN {X 0,Y 460.542,Z 400.615,A -85,B 0,C 180,E1 -7899.453,E2 -7899.453} C_VEL
LIN {X 0,Y 460.55,Z 400.614,A -85,B 0,C 180,E1 -7902.23,E2 -7902.23} C_VEL
LIN {X 0,Y 460.556,Z 400.617,A -85,B 0,C 180,E1 -7904.965,E2 -7904.965} C_VEL
LIN {X 0,Y 460.599,Z 400.606,A -85,B 0,C 180,E1 -7907.666,E2 -7907.666} C_VEL
LIN {X 0,Y 460.619,Z 400.605,A -85,B 0,C 180,E1 -7911.224,E2 -7911.224} C_VEL
LIN {X 0,Y 460.703,Z 400.594,A -85,B 0,C 180,E1 -7913.871,E2 -7913.871} C_VEL
LIN {X 0,Y 460.817,Z 400.579,A -85,B 0,C 180,E1 -7917.378,E2 -7917.378} C_VEL
LIN {X 0,Y 460.844,Z 400.578,A -85,B 0,C 180,E1 -7920,E2 -7920} C_VEL
LIN {X 0,Y 460.817,Z 400.585,A -85,B 0,C 180,E1 -7922.623,E2 -7922.623} C_VEL
LIN {X 0,Y 460.701,Z 400.598,A -85,B 0,C 180,E1 -7926.13,E2 -7926.13} C_VEL
LIN {X 0,Y 460.621,Z 400.607,A -85,B 0,C 180,E1 -7928.777,E2 -7928.777} C_VEL
LIN {X 0,Y 460.605,Z 400.612,A -85,B 0,C 180,E1 -7932.446,E2 -7932.446} C_VEL
LIN {X 0,Y 460.615,Z 400.609,A -85,B 0,C 180,E1 -7936.008,E2 -7936.008} C_VEL
LIN {X 0,Y 460.561,Z 400.612,A -85,B 0,C 180,E1 -7939.616,E2 -7939.616} C_VEL
LIN {X 0,Y 460.504,Z 400.623,A -85,B 0,C 180,E1 -7942.429,E2 -7942.429} C_VEL
LIN {X 0,Y 460.562,Z 400.615,A -85,B 0,C 180,E1 -7945.803,E2 -7945.803} C_VEL
LIN {X 0,Y 460.549,Z 400.618,A -85,B 0,C 180,E1 -7948.234,E2 -7948.234} C_VEL
LIN {X 0,Y 460.519,Z 400.617,A -85,B 0,C 180,E1 -7951.285,E2 -7951.285} C_VEL
LIN {X 0,Y 460.53,Z 400.618,A -85,B 0,C 180,E1 -7954.507,E2 -7954.507} C_VEL
LIN {X 0,Y 460.526,Z 400.623,A -85,B 0,C 180,E1 -7957.621,E2 -7957.621} C_VEL
LIN {X 0,Y 460.554,Z 400.62,A -85,B 0,C 180,E1 -7960.273,E2 -7960.273} C_VEL
LIN {X 0,Y 460.544,Z 400.722,A -85,B 0,C 180,E1 -7961.606,E2 -7961.606} C_VEL
LIN {X 0,Y 461.008,Z 403.951,A -85,B 0,C 180,E1 -7964.529,E2 -7964.529} C_VEL
LIN {X 0,Y 461.364,Z 406.889,A -85,B 0,C 180,E1 -7966.987,E2 -7966.987} C_VEL
LIN {X 0,Y 461.314,Z 410.337,A -85,B 0,C 180,E1 -7969.618,E2 -7969.618} C_VEL
LIN {X 0,Y 461.171,Z 414.265,A -85,B 0,C 180,E1 -7972.442,E2 -7972.442} C_VEL
LIN {X 0,Y 460.874,Z 419.064,A -85,B 0,C 180,E1 -7975.653,E2 -7975.653} C_VEL
LIN {X 0,Y 460.594,Z 423.925,A -85,B 0,C 180,E1 -7978.75,E2 -7978.75} C_VEL
LIN {X 0,Y 460.336,Z 428.898,A -85,B 0,C 180,E1 -7981.753,E2 -7981.753} C_VEL
LIN {X 0,Y 460.139,Z 433.934,A -85,B 0,C 180,E1 -7984.681,E2 -7984.681} C_VEL
LIN {X 0,Y 459.924,Z 439.034,A -85,B 0,C 180,E1 -7987.542,E2 -7987.542} C_VEL
LIN {X 0,Y 459.806,Z 444.195,A -85,B 0,C 180,E1 -7990.351,E2 -7990.351} C_VEL
LIN {X 0,Y 459.69,Z 449.389,A -85,B 0,C 180,E1 -7993.114,E2 -7993.114} C_VEL
LIN {X 0,Y 459.703,Z 451.831,A -85,B 0,C 180,E1 -7994.382,E2 -7994.382} C_VEL
LIN {X 0,Y 461.703,Z 463.325,A -85,B 0,C 180,E1 -7994.769,E2 -7994.769} C_VEL
LIN {X 0,Y 463.071,Z 473.552,A -85,B 0,C 180,E1 -7995.217,E2 -7995.217} C_VEL
LIN {X 0,Y 462.608,Z 485.37,A -85,B 0,C 180,E1 -7995.82,E2 -7995.82} C_VEL
LIN {X 0,Y 462.094,Z 496.771,A -85,B 0,C 180,E1 -7996.589,E2 -7996.589} C_VEL
LIN {X 0,Y 461.655,Z 505.812,A -85,B 0,C 180,E1 -7997.347,E2 -7997.347} C_VEL
LIN {X 0,Y 461.252,Z 513.683,A -85,B 0,C 180,E1 -7998.13,E2 -7998.13} C_VEL
LIN {X 0,Y 460.764,Z 522.823,A -85,B 0,C 180,E1 -7999.231,E2 -7999.231} C_VEL
LIN {X 0,Y 460.463,Z 529.026,A -85,B 0,C 180,E1 -8000.113,E2 -8000.113} C_VEL
LIN {X 0,Y 460.165,Z 535.565,A -85,B 0,C 180,E1 -8001.215,E2 -8001.215} C_VEL
LIN {X 0,Y 459.949,Z 540.066,A -85,B 0,C 180,E1 -8002.096,E2 -8002.096} C_VEL
LIN {X 0,Y 459.741,Z 545.557,A -85,B 0,C 180,E1 -8003.417,E2 -8003.417} C_VEL
LIN {X 0,Y 459.66,Z 549.879,A -85,B 0,C 180,E1 -8004.737,E2 -8004.737} C_VEL
LIN {X 0,Y 459.572,Z 552.242,A -85,B 0,C 180,E1 -8005.615,E2 -8005.615} C_VEL
LIN {X 0,Y 459.587,Z 554.04,A -85,B 0,C 180,E1 -8006.493,E2 -8006.493} C_VEL
LIN {X 0,Y 459.521,Z 556.48,A -85,B 0,C 180,E1 -8008.247,E2 -8008.247} C_VEL
LIN {X 0,Y 459.522,Z 557.068,A -85,B 0,C 180,E1 -8009.124,E2 -8009.124} C_VEL
LIN {X 0,Y 459.522,Z 557.068,A -85,B 0,C 180,E1 -8010.876,E2 -8010.876} C_VEL
LIN {X 0,Y 459.521,Z 556.48,A -85,B 0,C 180,E1 -8011.753,E2 -8011.753} C_VEL
LIN {X 0,Y 459.587,Z 554.04,A -85,B 0,C 180,E1 -8013.507,E2 -8013.507} C_VEL
LIN {X 0,Y 459.625,Z 551.094,A -85,B 0,C 180,E1 -8014.824,E2 -8014.824} C_VEL
LIN {X 0,Y 459.676,Z 547.108,A -85,B 0,C 180,E1 -8016.144,E2 -8016.144} C_VEL
LIN {X 0,Y 459.865,Z 541.981,A -85,B 0,C 180,E1 -8017.464,E2 -8017.464} C_VEL
LIN {X 0,Y 460.117,Z 536.72,A -85,B 0,C 180,E1 -8018.564,E2 -8018.564} C_VEL
LIN {X 0,Y 460.378,Z 530.402,A -85,B 0,C 180,E1 -8019.667,E2 -8019.667} C_VEL
LIN {X 0,Y 460.638,Z 524.449,A -85,B 0,C 180,E1 -8020.549,E2 -8020.549} C_VEL
LIN {X 0,Y 461.042,Z 517.522,A -85,B 0,C 180,E1 -8021.43,E2 -8021.43} C_VEL
LIN {X 0,Y 461.507,Z 509.342,A -85,B 0,C 180,E1 -8022.309,E2 -8022.309} C_VEL
LIN {X 0,Y 461.772,Z 502.214,A -85,B 0,C 180,E1 -8022.97,E2 -8022.97} C_VEL
LIN {X 0,Y 462.281,Z 492.108,A -85,B 0,C 180,E1 -8023.741,E2 -8023.741} C_VEL
LIN {X 0,Y 462.76,Z 482.348,A -85,B 0,C 180,E1 -8024.343,E2 -8024.343} C_VEL
LIN {X 0,Y 463.074,Z 473.552,A -85,B 0,C 180,E1 -8024.783,E2 -8024.783} C_VEL
LIN {X 0,Y 461.57,Z 462.623,A -85,B 0,C 180,E1 -8025.258,E2 -8025.258} C_VEL
LIN {X 0,Y 459.825,Z 453.022,A -85,B 0,C 180,E1 -8025.584,E2 -8025.584} C_VEL
LIN {X 0,Y 459.694,Z 451.796,A -85,B 0,C 180,E1 -8025.635,E2 -8025.635} C_VEL
LIN {X 0,Y 459.796,Z 445.907,A -85,B 0,C 180,E1 -8028.722,E2 -8028.722} C_VEL
LIN {X 0,Y 459.913,Z 440.741,A -85,B 0,C 180,E1 -8031.515,E2 -8031.515} C_VEL
LIN {X 0,Y 460.045,Z 435.624,A -85,B 0,C 180,E1 -8034.36,E2 -8034.36} C_VEL
LIN {X 0,Y 460.307,Z 429.839,A -85,B 0,C 180,E1 -8037.68,E2 -8037.68} C_VEL
LIN {X 0,Y 460.512,Z 425.566,A -85,B 0,C 180,E1 -8040.239,E2 -8040.239} C_VEL
LIN {X 0,Y 460.753,Z 420.656,A -85,B 0,C 180,E1 -8043.306,E2 -8043.306} C_VEL
LIN {X 0,Y 461.06,Z 415.838,A -85,B 0,C 180,E1 -8046.475,E2 -8046.475} C_VEL
LIN {X 0,Y 461.294,Z 411.134,A -85,B 0,C 180,E1 -8049.782,E2 -8049.782} C_VEL
LIN {X 0,Y 461.387,Z 408.054,A -85,B 0,C 180,E1 -8052.083,E2 -8052.083} C_VEL
LIN {X 0,Y 461.169,Z 405.067,A -85,B 0,C 180,E1 -8054.507,E2 -8054.507} C_VEL
LIN {X 0,Y 460.622,Z 401.326,A -85,B 0,C 180,E1 -8057.829,E2 -8057.829} C_VEL
LIN {X 0,Y 460.544,Z 400.72,A -85,B 0,C 180,E1 -8058.394,E2 -8058.394} C_VEL
LIN {X 0,Y 460.535,Z 400.619,A -85,B 0,C 180,E1 -8061.267,E2 -8061.267} C_VEL
LIN {X 0,Y 460.509,Z 400.624,A -85,B 0,C 180,E1 -8064.554,E2 -8064.554} C_VEL
LIN {X 0,Y 460.528,Z 400.619,A -85,B 0,C 180,E1 -8067.715,E2 -8067.715} C_VEL
LIN {X 0,Y 460.541,Z 400.614,A -85,B 0,C 180,E1 -8070.769,E2 -8070.769} C_VEL
LIN {X 0,Y 460.557,Z 400.617,A -85,B 0,C 180,E1 -8073.734,E2 -8073.734} C_VEL
LIN {X 0,Y 460.539,Z 400.614,A -85,B 0,C 180,E1 -8076.623,E2 -8076.623} C_VEL
LIN {X 0,Y 460.544,Z 400.617,A -85,B 0,C 180,E1 -8079.452,E2 -8079.452} C_VEL
LIN {X 0,Y 460.552,Z 400.614,A -85,B 0,C 180,E1 -8082.229,E2 -8082.229} C_VEL
LIN {X 0,Y 460.562,Z 400.611,A -85,B 0,C 180,E1 -8084.964,E2 -8084.964} C_VEL
LIN {X 0,Y 460.603,Z 400.606,A -85,B 0,C 180,E1 -8088.559,E2 -8088.559} C_VEL
LIN {X 0,Y 460.687,Z 400.597,A -85,B 0,C 180,E1 -8092.108,E2 -8092.108} C_VEL
LIN {X 0,Y 460.69,Z 400.595,A -85,B 0,C 180,E1 -8094.748,E2 -8094.748} C_VEL
LIN {X 0,Y 460.817,Z 400.585,A -85,B 0,C 180,E1 -8097.377,E2 -8097.377} C_VEL
LIN {X 0,Y 460.844,Z 400.578,A -85,B 0,C 180,E1 -8100,E2 -8100} C_VEL
LIN {X 0,Y 460.817,Z 400.579,A -85,B 0,C 180,E1 -8102.622,E2 -8102.622} C_VEL
LIN {X 0,Y 460.703,Z 400.594,A -85,B 0,C 180,E1 -8106.129,E2 -8106.129} C_VEL
LIN {X 0,Y 460.62,Z 400.605,A -85,B 0,C 180,E1 -8108.776,E2 -8108.776} C_VEL
LIN {X 0,Y 460.604,Z 400.606,A -85,B 0,C 180,E1 -8112.445,E2 -8112.445} C_VEL
LIN {X 0,Y 460.59,Z 400.608,A -85,B 0,C 180,E1 -8115.997,E2 -8115.997} C_VEL
LIN {X 0,Y 460.561,Z 400.616,A -85,B 0,C 180,E1 -8118.902,E2 -8118.902} C_VEL
LIN {X 0,Y 460.506,Z 400.621,A -85,B 0,C 180,E1 -8121.486,E2 -8121.486} C_VEL
LIN {X 0,Y 460.533,Z 400.615,A -85,B 0,C 180,E1 -8124.332,E2 -8124.332} C_VEL
LIN {X 0,Y 460.575,Z 400.614,A -85,B 0,C 180,E1 -8127.243,E2 -8127.243} C_VEL
LIN {X 0,Y 460.518,Z 400.617,A -85,B 0,C 180,E1 -8130.239,E2 -8130.239} C_VEL
LIN {X 0,Y 460.52,Z 400.619,A -85,B 0,C 180,E1 -8133.325,E2 -8133.325} C_VEL
LIN {X 0,Y 460.471,Z 400.626,A -85,B 0,C 180,E1 -8136.529,E2 -8136.529} C_VEL
LIN {X 0,Y 460.57,Z 400.61,A -85,B 0,C 180,E1 -8139.858,E2 -8139.858} C_VEL
LIN {X 0,Y 460.535,Z 400.62,A -85,B 0,C 180,E1 -8142.905,E2 -8142.905} C_VEL
LIN {X 0,Y 460.511,Z 400.617,A -85,B 0,C 180,E1 -8145.83,E2 -8145.83} C_VEL
LIN {X 0,Y 460.526,Z 400.619,A -85,B 0,C 180,E1 -8148.989,E2 -8148.989} C_VEL
LIN {X 0,Y 460.519,Z 400.617,A -85,B 0,C 180,E1 -8151.267,E2 -8151.267} C_VEL
LIN {X 0,Y 460.507,Z 400.626,A -85,B 0,C 180,E1 -8154.555,E2 -8154.555} C_VEL
LIN {X 0,Y 460.526,Z 400.616,A -85,B 0,C 180,E1 -8157.716,E2 -8157.716} C_VEL
LIN {X 0,Y 460.534,Z 400.618,A -85,B 0,C 180,E1 -8160.769,E2 -8160.769} C_VEL
LIN {X 0,Y 460.563,Z 400.611,A -85,B 0,C 180,E1 -8163.735,E2 -8163.735} C_VEL
LIN {X 0,Y 460.541,Z 400.618,A -85,B 0,C 180,E1 -8166.624,E2 -8166.624} C_VEL
LIN {X 0,Y 460.546,Z 400.613,A -85,B 0,C 180,E1 -8169.453,E2 -8169.453} C_VEL
LIN {X 0,Y 460.555,Z 400.62,A -85,B 0,C 180,E1 -8172.23,E2 -8172.23} C_VEL
LIN {X 0,Y 460.561,Z 400.615,A -85,B 0,C 180,E1 -8174.965,E2 -8174.965} C_VEL
LIN {X 0,Y 460.608,Z 400.612,A -85,B 0,C 180,E1 -8178.559,E2 -8178.559} C_VEL
LIN {X 0,Y 460.574,Z 400.613,A -85,B 0,C 180,E1 -8179.233,E2 -8179.233} C_VEL
LIN {X 0,Y 459.919,Z 400.698,A -85,B 0,C 180,E1 -8179.963,E2 -8179.963} C_VEL
LIN {X 0,Y 457.102,Z 401.047,A -85,B 0,C 180,E1 -8181.15,E2 -8181.15} C_VEL
LIN {X 0,Y 454.722,Z 401.345,A -85,B 0,C 180,E1 -8182.107,E2 -8182.107} C_VEL
LIN {X 0,Y 453.711,Z 401.468,A -85,B 0,C 180,E1 -8182.846,E2 -8182.846} C_VEL
LIN {X 0,Y 453.634,Z 401.477,A -85,B 0,C 180,E1 -8183.096,E2 -8183.096} C_VEL
LIN {X 0,Y 453.668,Z 401.475,A -85,B 0,C 180,E1 -8184.667,E2 -8184.667} C_VEL
LIN {X 0,Y 453.762,Z 401.462,A -85,B 0,C 180,E1 -8187.337,E2 -8187.337} C_VEL
LIN {X 0,Y 453.821,Z 401.459,A -85,B 0,C 180,E1 -8190,E2 -8190} C_VEL
LIN {X 0,Y 453.762,Z 401.462,A -85,B 0,C 180,E1 -8192.663,E2 -8192.663} C_VEL
LIN {X 0,Y 453.675,Z 401.475,A -85,B 0,C 180,E1 -8196.225,E2 -8196.225} C_VEL
LIN {X 0,Y 453.589,Z 401.484,A -85,B 0,C 180,E1 -8198.913,E2 -8198.913} C_VEL
LIN {X 0,Y 453.559,Z 401.486,A -85,B 0,C 180,E1 -8202.529,E2 -8202.529} C_VEL
LIN {X 0,Y 453.54,Z 401.491,A -85,B 0,C 180,E1 -8206.196,E2 -8206.196} C_VEL
LIN {X 0,Y 453.515,Z 401.493,A -85,B 0,C 180,E1 -8209.04,E2 -8209.04} C_VEL
LIN {X 0,Y 453.471,Z 401.5,A -85,B 0,C 180,E1 -8211.836,E2 -8211.836} C_VEL
LIN {X 0,Y 453.509,Z 401.49,A -85,B 0,C 180,E1 -8214.734,E2 -8214.734} C_VEL
LIN {X 0,Y 453.532,Z 401.489,A -85,B 0,C 180,E1 -8217.961,E2 -8217.961} C_VEL
LIN {X 0,Y 453.461,Z 401.503,A -85,B 0,C 180,E1 -8221.525,E2 -8221.525} C_VEL
LIN {X 0,Y 453.483,Z 401.494,A -85,B 0,C 180,E1 -8224.777,E2 -8224.777} C_VEL
LIN {X 0,Y 453.466,Z 401.495,A -85,B 0,C 180,E1 -8228.31,E2 -8228.31} C_VEL
LIN {X 0,Y 453.487,Z 401.493,A -85,B 0,C 180,E1 -8230.609,E2 -8230.609} C_VEL
LIN {X 0,Y 453.456,Z 401.503,A -85,B 0,C 180,E1 -8233.245,E2 -8233.245} C_VEL
LIN {X 0,Y 453.466,Z 401.497,A -85,B 0,C 180,E1 -8235.78,E2 -8235.78} C_VEL
LIN {X 0,Y 453.473,Z 401.494,A -85,B 0,C 180,E1 -8238.209,E2 -8238.209} C_VEL
LIN {X 0,Y 453.486,Z 401.495,A -85,B 0,C 180,E1 -8240.793,E2 -8240.793} C_VEL
LIN {X 0,Y 453.448,Z 401.497,A -85,B 0,C 180,E1 -8243.917,E2 -8243.917} C_VEL
LIN {X 0,Y 453.474,Z 401.501,A -85,B 0,C 180,E1 -8247.151,E2 -8247.151} C_VEL
LIN {X 0,Y 453.505,Z 401.49,A -85,B 0,C 180,E1 -8250.271,E2 -8250.271} C_VEL
LIN {X 0,Y 453.505,Z 401.494,A -85,B 0,C 180,E1 -8253.294,E2 -8253.294} C_VEL
LIN {X 0,Y 453.494,Z 401.492,A -85,B 0,C 180,E1 -8256.239,E2 -8256.239} C_VEL
LIN {X 0,Y 453.473,Z 401.499,A -85,B 0,C 180,E1 -8259.118,E2 -8259.118} C_VEL
LIN {X 0,Y 453.502,Z 401.49,A -85,B 0,C 180,E1 -8261.945,E2 -8261.945} C_VEL
LIN {X 0,Y 453.53,Z 401.494,A -85,B 0,C 180,E1 -8264.727,E2 -8264.727} C_VEL
LIN {X 0,Y 453.554,Z 401.484,A -85,B 0,C 180,E1 -8267.471,E2 -8267.471} C_VEL
LIN {X 0,Y 453.583,Z 401.483,A -85,B 0,C 180,E1 -8271.087,E2 -8271.087} C_VEL
LIN {X 0,Y 453.67,Z 401.469,A -85,B 0,C 180,E1 -8273.775,E2 -8273.775} C_VEL
LIN {X 0,Y 453.757,Z 401.459,A -85,B 0,C 180,E1 -8277.337,E2 -8277.337} C_VEL
LIN {X 0,Y 453.814,Z 401.453,A -85,B 0,C 180,E1 -8280,E2 -8280} C_VEL
LIN {X 0,Y 453.757,Z 401.464,A -85,B 0,C 180,E1 -8282.664,E2 -8282.664} C_VEL
LIN {X 0,Y 453.669,Z 401.475,A -85,B 0,C 180,E1 -8286.226,E2 -8286.226} C_VEL
LIN {X 0,Y 453.585,Z 401.482,A -85,B 0,C 180,E1 -8288.914,E2 -8288.914} C_VEL
LIN {X 0,Y 453.555,Z 401.489,A -85,B 0,C 180,E1 -8292.53,E2 -8292.53} C_VEL
LIN {X 0,Y 453.549,Z 401.492,A -85,B 0,C 180,E1 -8296.196,E2 -8296.196} C_VEL
LIN {X 0,Y 453.513,Z 401.489,A -85,B 0,C 180,E1 -8299.041,E2 -8299.041} C_VEL
LIN {X 0,Y 453.47,Z 401.498,A -85,B 0,C 180,E1 -8301.837,E2 -8301.837} C_VEL
LIN {X 0,Y 453.508,Z 401.491,A -85,B 0,C 180,E1 -8304.735,E2 -8304.735} C_VEL
LIN {X 0,Y 453.527,Z 401.494,A -85,B 0,C 180,E1 -8307.961,E2 -8307.961} C_VEL
LIN {X 0,Y 453.478,Z 401.494,A -85,B 0,C 180,E1 -8310.76,E2 -8310.76} C_VEL
LIN {X 0,Y 453.473,Z 401.501,A -85,B 0,C 180,E1 -8313.913,E2 -8313.913} C_VEL
LIN {X 0,Y 453.467,Z 401.499,A -85,B 0,C 180,E1 -8317.189,E2 -8317.189} C_VEL
LIN {X 0,Y 453.524,Z 401.494,A -85,B 0,C 180,E1 -8319.447,E2 -8319.447} C_VEL
LIN {X 0,Y 453.513,Z 401.496,A -85,B 0,C 180,E1 -8320.607,E2 -8320.607} C_VEL
LIN {X 0,Y 453.607,Z 402.281,A -85,B 0,C 180,E1 -8321.955,E2 -8321.955} C_VEL
LIN {X 0,Y 454.153,Z 406.086,A -85,B 0,C 180,E1 -8325.386,E2 -8325.386} C_VEL
LIN {X 0,Y 454.381,Z 409.2,A -85,B 0,C 180,E1 -8327.939,E2 -8327.939} C_VEL
LIN {X 0,Y 454.238,Z 412.81,A -85,B 0,C 180,E1 -8330.679,E2 -8330.679} C_VEL
LIN {X 0,Y 454.018,Z 416.94,A -85,B 0,C 180,E1 -8333.605,E2 -8333.605} C_VEL
LIN {X 0,Y 453.725,Z 421.658,A -85,B 0,C 180,E1 -8336.766,E2 -8336.766} C_VEL
LIN {X 0,Y 453.506,Z 425.538,A -85,B 0,C 180,E1 -8339.243,E2 -8339.243} C_VEL
LIN {X 0,Y 453.272,Z 430.504,A -85,B 0,C 180,E1 -8342.281,E2 -8342.281} C_VEL
LIN {X 0,Y 453.009,Z 435.541,A -85,B 0,C 180,E1 -8345.237,E2 -8345.237} C_VEL
LIN {X 0,Y 452.839,Z 441.507,A -85,B 0,C 180,E1 -8348.622,E2 -8348.622} C_VEL
LIN {X 0,Y 452.659,Z 447.508,A -85,B 0,C 180,E1 -8351.91,E2 -8351.91} C_VEL
LIN {X 0,Y 452.616,Z 451.668,A -85,B 0,C 180,E1 -8354.131,E2 -8354.131} C_VEL
LIN {X 0,Y 454.553,Z 462.951,A -85,B 0,C 180,E1 -8354.518,E2 -8354.518} C_VEL
LIN {X 0,Y 456.069,Z 473.351,A -85,B 0,C 180,E1 -8354.985,E2 -8354.985} C_VEL
LIN {X 0,Y 455.806,Z 483.158,A -85,B 0,C 180,E1 -8355.49,E2 -8355.49} C_VEL
LIN {X 0,Y 455.247,Z 495.154,A -85,B 0,C 180,E1 -8356.27,E2 -8356.27} C_VEL
LIN {X 0,Y 454.671,Z 505.973,A -85,B 0,C 180,E1 -8357.186,E2 -8357.186} C_VEL
LIN {X 0,Y 454.281,Z 513.485,A -85,B 0,C 180,E1 -8357.945,E2 -8357.945} C_VEL
LIN {X 0,Y 453.734,Z 522.625,A -85,B 0,C 180,E1 -8359.062,E2 -8359.062} C_VEL
LIN {X 0,Y 453.438,Z 528.828,A -85,B 0,C 180,E1 -8359.958,E2 -8359.958} C_VEL
LIN {X 0,Y 453.115,Z 535.367,A -85,B 0,C 180,E1 -8361.077,E2 -8361.077} C_VEL
LIN {X 0,Y 452.893,Z 539.868,A -85,B 0,C 180,E1 -8361.972,E2 -8361.972} C_VEL
LIN {X 0,Y 452.651,Z 545.513,A -85,B 0,C 180,E1 -8363.358,E2 -8363.358} C_VEL
LIN {X 0,Y 452.575,Z 549.681,A -85,B 0,C 180,E1 -8364.654,E2 -8364.654} C_VEL
LIN {X 0,Y 452.494,Z 552.045,A -85,B 0,C 180,E1 -8365.546,E2 -8365.546} C_VEL
LIN {X 0,Y 452.484,Z 553.842,A -85,B 0,C 180,E1 -8366.438,E2 -8366.438} C_VEL
LIN {X 0,Y 452.437,Z 556.283,A -85,B 0,C 180,E1 -8368.22,E2 -8368.22} C_VEL
LIN {X 0,Y 452.429,Z 556.871,A -85,B 0,C 180,E1 -8369.11,E2 -8369.11} C_VEL
LIN {X 0,Y 452.429,Z 556.871,A -85,B 0,C 180,E1 -8370.89,E2 -8370.89} C_VEL
LIN {X 0,Y 452.437,Z 556.283,A -85,B 0,C 180,E1 -8371.78,E2 -8371.78} C_VEL
LIN {X 0,Y 452.484,Z 553.842,A -85,B 0,C 180,E1 -8373.562,E2 -8373.562} C_VEL
LIN {X 0,Y 452.553,Z 550.897,A -85,B 0,C 180,E1 -8374.9,E2 -8374.9} C_VEL
LIN {X 0,Y 452.605,Z 546.911,A -85,B 0,C 180,E1 -8376.24,E2 -8376.24} C_VEL
LIN {X 0,Y 452.814,Z 541.784,A -85,B 0,C 180,E1 -8377.581,E2 -8377.581} C_VEL
LIN {X 0,Y 453.058,Z 536.522,A -85,B 0,C 180,E1 -8378.699,E2 -8378.699} C_VEL
LIN {X 0,Y 453.35,Z 530.204,A -85,B 0,C 180,E1 -8379.818,E2 -8379.818} C_VEL
LIN {X 0,Y 453.629,Z 524.251,A -85,B 0,C 180,E1 -8380.714,E2 -8380.714} C_VEL
LIN {X 0,Y 454.045,Z 517.324,A -85,B 0,C 180,E1 -8381.608,E2 -8381.608} C_VEL
LIN {X 0,Y 454.533,Z 509.143,A -85,B 0,C 180,E1 -8382.501,E2 -8382.501} C_VEL
LIN {X 0,Y 454.886,Z 500.539,A -85,B 0,C 180,E1 -8383.294,E2 -8383.294} C_VEL
LIN {X 0,Y 455.385,Z 491.911,A -85,B 0,C 180,E1 -8383.954,E2 -8383.954} C_VEL
LIN {X 0,Y 455.841,Z 482.15,A -85,B 0,C 180,E1 -8384.566,E2 -8384.566} C_VEL
LIN {X 0,Y 456.065,Z 473.351,A -85,B 0,C 180,E1 -8385.015,E2 -8385.015} C_VEL
LIN {X 0,Y 454.558,Z 462.97,A -85,B 0,C 180,E1 -8385.481,E2 -8385.481} C_VEL
LIN {X 0,Y 452.743,Z 452.863,A -85,B 0,C 180,E1 -8385.833,E2 -8385.833} C_VEL
LIN {X 0,Y 452.632,Z 451.679,A -85,B 0,C 180,E1 -8385.863,E2 -8385.863} C_VEL
LIN {X 0,Y 452.723,Z 445.769,A -85,B 0,C 180,E1 -8389.026,E2 -8389.026} C_VEL
LIN {X 0,Y 452.84,Z 440.631,A -85,B 0,C 180,E1 -8391.868,E2 -8391.868} C_VEL
LIN {X 0,Y 453.009,Z 435.538,A -85,B 0,C 180,E1 -8394.763,E2 -8394.763} C_VEL
LIN {X 0,Y 453.259,Z 430.209,A -85,B 0,C 180,E1 -8397.894,E2 -8397.894} C_VEL
LIN {X 0,Y 453.506,Z 425.536,A -85,B 0,C 180,E1 -8400.757,E2 -8400.757} C_VEL
LIN {X 0,Y 453.768,Z 420.651,A -85,B 0,C 180,E1 -8403.887,E2 -8403.887} C_VEL
LIN {X 0,Y 454.068,Z 415.863,A -85,B 0,C 180,E1 -8407.13,E2 -8407.13} C_VEL
LIN {X 0,Y 454.241,Z 412.72,A -85,B 0,C 180,E1 -8409.371,E2 -8409.371} C_VEL
LIN {X 0,Y 454.381,Z 409.163,A -85,B 0,C 180,E1 -8412.061,E2 -8412.061} C_VEL
LIN {X 0,Y 454.15,Z 406.08,A -85,B 0,C 180,E1 -8414.614,E2 -8414.614} C_VEL
LIN {X 0,Y 453.607,Z 402.28,A -85,B 0,C 180,E1 -8418.045,E2 -8418.045} C_VEL
LIN {X 0,Y 453.513,Z 401.495,A -85,B 0,C 180,E1 -8419.405,E2 -8419.405} C_VEL
LIN {X 0,Y 453.472,Z 401.502,A -85,B 0,C 180,E1 -8422.222,E2 -8422.222} C_VEL
LIN {X 0,Y 453.485,Z 401.497,A -85,B 0,C 180,E1 -8425.221,E2 -8425.221} C_VEL
LIN {X 0,Y 453.463,Z 401.497,A -85,B 0,C 180,E1 -8428.473,E2 -8428.473} C_VEL
LIN {X 0,Y 453.51,Z 401.49,A -85,B 0,C 180,E1 -8431.288,E2 -8431.288} C_VEL
LIN {X 0,Y 453.518,Z 401.491,A -85,B 0,C 180,E1 -8434.284,E2 -8434.284} C_VEL
LIN {X 0,Y 453.473,Z 401.495,A -85,B 0,C 180,E1 -8437.203,E2 -8437.203} C_VEL
LIN {X 0,Y 453.497,Z 401.495,A -85,B 0,C 180,E1 -8440.065,E2 -8440.065} C_VEL
LIN {X 0,Y 453.502,Z 401.49,A -85,B 0,C 180,E1 -8442.875,E2 -8442.875} C_VEL
LIN {X 0,Y 453.507,Z 401.497,A -85,B 0,C 180,E1 -8445.643,E2 -8445.643} C_VEL
LIN {X 0,Y 453.552,Z 401.485,A -85,B 0,C 180,E1 -8448.378,E2 -8448.378} C_VEL
LIN {X 0,Y 453.644,Z 401.476,A -85,B 0,C 180,E1 -8451.985,E2 -8451.985} C_VEL
LIN {X 0,Y 453.663,Z 401.47,A -85,B 0,C 180,E1 -8454.666,E2 -8454.666} C_VEL
LIN {X 0,Y 453.757,Z 401.464,A -85,B 0,C 180,E1 -8457.336,E2 -8457.336} C_VEL
LIN {X 0,Y 453.814,Z 401.453,A -85,B 0,C 180,E1 -8460,E2 -8460} C_VEL
LIN {X 0,Y 453.757,Z 401.459,A -85,B 0,C 180,E1 -8462.663,E2 -8462.663} C_VEL
LIN {X 0,Y 453.67,Z 401.469,A -85,B 0,C 180,E1 -8466.225,E2 -8466.225} C_VEL
LIN {X 0,Y 453.583,Z 401.483,A -85,B 0,C 180,E1 -8468.913,E2 -8468.913} C_VEL
LIN {X 0,Y 453.554,Z 401.484,A -85,B 0,C 180,E1 -8472.529,E2 -8472.529} C_VEL
LIN {X 0,Y 453.535,Z 401.486,A -85,B 0,C 180,E1 -8476.196,E2 -8476.196} C_VEL
LIN {X 0,Y 453.511,Z 401.496,A -85,B 0,C 180,E1 -8479.041,E2 -8479.041} C_VEL
LIN {X 0,Y 453.467,Z 401.495,A -85,B 0,C 180,E1 -8481.836,E2 -8481.836} C_VEL
LIN {X 0,Y 453.505,Z 401.494,A -85,B 0,C 180,E1 -8484.734,E2 -8484.734} C_VEL
LIN {X 0,Y 453.53,Z 401.487,A -85,B 0,C 180,E1 -8487.961,E2 -8487.961} C_VEL
LIN {X 0,Y 453.474,Z 401.499,A -85,B 0,C 180,E1 -8490.759,E2 -8490.759} C_VEL
LIN {X 0,Y 453.469,Z 401.494,A -85,B 0,C 180,E1 -8493.913,E2 -8493.913} C_VEL
LIN {X 0,Y 453.463,Z 401.499,A -85,B 0,C 180,E1 -8497.188,E2 -8497.188} C_VEL
LIN {X 0,Y 453.525,Z 401.489,A -85,B 0,C 180,E1 -8499.445,E2 -8499.445} C_VEL
LIN {X 0,Y 453.484,Z 401.497,A -85,B 0,C 180,E1 -8502.992,E2 -8502.992} C_VEL
LIN {X 0,Y 453.465,Z 401.495,A -85,B 0,C 180,E1 -8505.78,E2 -8505.78} C_VEL
LIN {X 0,Y 453.474,Z 401.496,A -85,B 0,C 180,E1 -8508.21,E2 -8508.21} C_VEL
LIN {X 0,Y 453.508,Z 401.496,A -85,B 0,C 180,E1 -8510.79,E2 -8510.79} C_VEL
LIN {X 0,Y 453.45,Z 401.498,A -85,B 0,C 180,E1 -8513.918,E2 -8513.918} C_VEL
LIN {X 0,Y 453.477,Z 401.495,A -85,B 0,C 180,E1 -8517.152,E2 -8517.152} C_VEL
LIN {X 0,Y 453.469,Z 401.499,A -85,B 0,C 180,E1 -8520.269,E2 -8520.269} C_VEL
LIN {X 0,Y 453.508,Z 401.49,A -85,B 0,C 180,E1 -8523.295,E2 -8523.295} C_VEL
LIN {X 0,Y 453.499,Z 401.497,A -85,B 0,C 180,E1 -8526.239,E2 -8526.239} C_VEL
LIN {X 0,Y 453.478,Z 401.495,A -85,B 0,C 180,E1 -8529.118,E2 -8529.118} C_VEL
LIN {X 0,Y 453.507,Z 401.496,A -85,B 0,C 180,E1 -8531.945,E2 -8531.945} C_VEL
LIN {X 0,Y 453.535,Z 401.491,A -85,B 0,C 180,E1 -8534.727,E2 -8534.727} C_VEL
LIN {X 0,Y 453.556,Z 401.49,A -85,B 0,C 180,E1 -8538.379,E2 -8538.379} C_VEL
LIN {X 0,Y 453.648,Z 401.478,A -85,B 0,C 180,E1 -8541.985,E2 -8541.985} C_VEL
LIN {X 0,Y 453.634,Z 401.477,A -85,B 0,C 180,E1 -8543.096,E2 -8543.096} C_VEL
LIN {X 0,Y 452.949,Z 401.566,A -85,B 0,C 180,E1 -8543.837,E2 -8543.837} C_VEL
LIN {X 0,Y 450,Z 401.931,A -85,B 0,C 180,E1 -8545.038,E2 -8545.038} C_VEL
LIN {X 0,Y 447.578,Z 402.235,A -85,B 0,C 180,E1 -8546.008,E2 -8546.008} C_VEL
LIN {X 0,Y 446.641,Z 402.349,A -85,B 0,C 180,E1 -8546.758,E2 -8546.758} C_VEL
LIN {X 0,Y 446.622,Z 402.351,A -85,B 0,C 180,E1 -8547.011,E2 -8547.011} C_VEL
LIN {X 0,Y 446.791,Z 402.334,A -85,B 0,C 180,E1 -8550,E2 -8550} C_VEL
LIN {X 0,Y 446.706,Z 402.341,A -85,B 0,C 180,E1 -8552.705,E2 -8552.705} C_VEL
LIN {X 0,Y 446.644,Z 402.35,A -85,B 0,C 180,E1 -8556.324,E2 -8556.324} C_VEL
LIN {X 0,Y 446.534,Z 402.363,A -85,B 0,C 180,E1 -8559.055,E2 -8559.055} C_VEL
LIN {X 0,Y 446.517,Z 402.363,A -85,B 0,C 180,E1 -8562.73,E2 -8562.73} C_VEL
LIN {X 0,Y 446.492,Z 402.369,A -85,B 0,C 180,E1 -8566.228,E2 -8566.228} C_VEL
LIN {X 0,Y 446.465,Z 402.373,A -85,B 0,C 180,E1 -8569.303,E2 -8569.303} C_VEL
LIN {X 0,Y 446.413,Z 402.375,A -85,B 0,C 180,E1 -8572.199,E2 -8572.199} C_VEL
LIN {X 0,Y 446.453,Z 402.371,A -85,B 0,C 180,E1 -8575.152,E2 -8575.152} C_VEL
LIN {X 0,Y 446.479,Z 402.366,A -85,B 0,C 180,E1 -8578.178,E2 -8578.178} C_VEL
LIN {X 0,Y 446.414,Z 402.377,A -85,B 0,C 180,E1 -8581.775,E2 -8581.775} C_VEL
LIN {X 0,Y 446.424,Z 402.372,A -85,B 0,C 180,E1 -8584.523,E2 -8584.523} C_VEL
LIN {X 0,Y 446.423,Z 402.373,A -85,B 0,C 180,E1 -8588.082,E2 -8588.082} C_VEL
LIN {X 0,Y 446.421,Z 402.375,A -85,B 0,C 180,E1 -8590.918,E2 -8590.918} C_VEL
LIN {X 0,Y 446.415,Z 402.375,A -85,B 0,C 180,E1 -8593.843,E2 -8593.843} C_VEL
LIN {X 0,Y 446.413,Z 402.374,A -85,B 0,C 180,E1 -8596.4,E2 -8596.4} C_VEL
LIN {X 0,Y 446.435,Z 402.372,A -85,B 0,C 180,E1 -8599.802,E2 -8599.802} C_VEL
LIN {X 0,Y 446.419,Z 402.373,A -85,B 0,C 180,E1 -8602.123,E2 -8602.123} C_VEL
LIN {X 0,Y 446.422,Z 402.375,A -85,B 0,C 180,E1 -8605.477,E2 -8605.477} C_VEL
LIN {X 0,Y 446.411,Z 402.377,A -85,B 0,C 180,E1 -8608.7,E2 -8608.7} C_VEL
LIN {X 0,Y 446.475,Z 402.366,A -85,B 0,C 180,E1 -8611.821,E2 -8611.821} C_VEL
LIN {X 0,Y 446.449,Z 402.376,A -85,B 0,C 180,E1 -8614.848,E2 -8614.848} C_VEL
LIN {X 0,Y 446.438,Z 402.371,A -85,B 0,C 180,E1 -8618.245,E2 -8618.245} C_VEL
LIN {X 0,Y 446.448,Z 402.369,A -85,B 0,C 180,E1 -8621.649,E2 -8621.649} C_VEL
LIN {X 0,Y 446.498,Z 402.367,A -85,B 0,C 180,E1 -8624.48,E2 -8624.48} C_VEL
LIN {X 0,Y 446.506,Z 402.363,A -85,B 0,C 180,E1 -8627.384,E2 -8627.384} C_VEL
LIN {X 0,Y 446.529,Z 402.363,A -85,B 0,C 180,E1 -8630.945,E2 -8630.945} C_VEL
LIN {X 0,Y 446.639,Z 402.345,A -85,B 0,C 180,E1 -8633.677,E2 -8633.677} C_VEL
LIN {X 0,Y 446.701,Z 402.338,A -85,B 0,C 180,E1 -8637.295,E2 -8637.295} C_VEL
LIN {X 0,Y 446.784,Z 402.329,A -85,B 0,C 180,E1 -8640.001,E2 -8640.001} C_VEL
LIN {X 0,Y 446.701,Z 402.343,A -85,B 0,C 180,E1 -8642.706,E2 -8642.706} C_VEL
LIN {X 0,Y 446.638,Z 402.352,A -85,B 0,C 180,E1 -8646.324,E2 -8646.324} C_VEL
LIN {X 0,Y 446.53,Z 402.36,A -85,B 0,C 180,E1 -8649.056,E2 -8649.056} C_VEL
LIN {X 0,Y 446.514,Z 402.364,A -85,B 0,C 180,E1 -8652.73,E2 -8652.73} C_VEL
LIN {X 0,Y 446.512,Z 402.369,A -85,B 0,C 180,E1 -8656.239,E2 -8656.239} C_VEL
LIN {X 0,Y 446.462,Z 402.367,A -85,B 0,C 180,E1 -8659.304,E2 -8659.304} C_VEL
LIN {X 0,Y 446.412,Z 402.381,A -85,B 0,C 180,E1 -8662.2,E2 -8662.2} C_VEL
LIN {X 0,Y 446.451,Z 402.369,A -85,B 0,C 180,E1 -8665.153,E2 -8665.153} C_VEL
